    |   movel([0.065962, -1.378345, -2.576120, -0.757924, 1.570796, 1.636759],accel_mss,speed_ms,0,blend_radius_m)
    |   speed_ms = 0.007
    |   movel([0.065737, -1.378110, -2.576285, -0.757994, 1.570796, 1.636533],accel_mss,speed_ms,0,blend_radius_m)
    |   movel([0.065748, -1.377418, -2.576770, -0.758201, 1.570796, 1.636545],accel_mss,speed_ms,0,blend_radius_m)
    |   movel([0.065782, -1.376692, -2.577278, -0.758419, 1.570796, 1.636578],accel_mss,speed_ms,0,blend_radius_m)
    |   movel([0.066186, -1.376388, -2.577490, -0.758511, 1.570796, 1.636982],accel_mss,speed_ms,0,blend_radius_m)
    |   movel([0.067252, -1.376135, -2.577667, -0.758587, 1.570796, 1.638048],accel_mss,speed_ms,0,blend_radius_m)
    |   movel([0.068316, -1.375910, -2.577824, -0.758655, 1.570796, 1.639113],accel_mss,speed_ms,0,blend_radius_m)
    |   movel([0.068585, -1.375943, -2.577801, -0.758645, 1.570796, 1.639381],accel_mss,speed_ms,0,blend_radius_m)
    |   movel([0.068684, -1.376248, -2.577588, -0.758553, 1.570796, 1.639480],accel_mss,speed_ms,0,blend_radius_m)
    |   movel([0.068626, -1.376569, -2.577364, -0.758456, 1.570796, 1.639422],accel_mss,speed_ms,0,blend_radius_m)
    |   movel([0.068470, -1.377126, -2.576974, -0.758289, 1.570796, 1.639267],accel_mss,speed_ms,0,blend_radius_m)
    |   movel([0.068277, -1.377389, -2.576790, -0.758210, 1.570796, 1.639073],accel_mss,speed_ms,0,blend_radius_m)
    |   movel([0.067750, -1.377691, -2.576579, -0.758120, 1.570796, 1.638546],accel_mss,speed_ms,0,blend_radius_m)
    |   movel([0.067148, -1.377954, -2.576394, -0.758041, 1.570796, 1.637944],accel_mss,speed_ms,0,blend_radius_m)
    |   movel([0.066517, -1.378181, -2.576235, -0.757973, 1.570796, 1.637313],accel_mss,speed_ms,0,blend_radius_m)
    |   movel([0.065962, -1.378345, -2.576120, -0.757924, 1.570796, 1.636759],accel_mss,speed_ms,0,blend_radius_m)
    |   speed_ms = 0.003
    |   movel([0.065962, -1.365252, -2.570091, -0.777046, 1.570796, 1.636759],accel_mss,speed_ms,0,blend_radius_m)
    |   speed_ms = 1.000
    |   movel([0.065962, -1.340154, -2.557638, -0.814597, 1.570796, 1.636759],accel_mss,speed_ms,0,blend_radius_m)
    |   movel([0.067314, -1.337303, -2.559523, -0.815563, 1.570796, 1.638110],accel_mss,speed_ms,0,blend_radius_m)
    |   movel([0.067314, -1.362450, -2.572012, -0.777926, 1.570796, 1.638110],accel_mss,speed_ms,0,blend_radius_m)
    |   speed_ms = 0.003
    |   movel([0.067314, -1.372257, -2.576561, -0.763571, 1.570796, 1.638110],accel_mss,speed_ms,0,blend_radius_m)
    |   speed_ms = 0.007
    |   movel([0.067188, -1.372005, -2.576736, -0.763648, 1.570796, 1.637984],accel_mss,speed_ms,0,blend_radius_m)
    |   movel([0.067191, -1.371585, -2.577027, -0.763777, 1.570796, 1.637988],accel_mss,speed_ms,0,blend_radius_m)
    |   movel([0.067248, -1.370744, -2.577609, -0.764035, 1.570796, 1.638044],accel_mss,speed_ms,0,blend_radius_m)
    |   movel([0.067309, -1.370030, -2.578103, -0.764256, 1.570796, 1.638105],accel_mss,speed_ms,0,blend_radius_m)
    |   movel([0.067374, -1.369514, -2.578460, -0.764415, 1.570796, 1.638171],accel_mss,speed_ms,0,blend_radius_m)
    |   movel([0.067446, -1.369137, -2.578720, -0.764532, 1.570796, 1.638242],accel_mss,speed_ms,0,blend_radius_m)
    |   movel([0.067665, -1.368841, -2.578924, -0.764624, 1.570796, 1.638462],accel_mss,speed_ms,0,blend_radius_m)
    |   movel([0.067820, -1.368984, -2.578825, -0.764580, 1.570796, 1.638616],accel_mss,speed_ms,0,blend_radius_m)
    |   movel([0.067982, -1.369133, -2.578722, -0.764534, 1.570796, 1.638778],accel_mss,speed_ms,0,blend_radius_m)
    |   movel([0.067952, -1.369386, -2.578548, -0.764455, 1.570796, 1.638748],accel_mss,speed_ms,0,blend_radius_m)
    |   movel([0.067835, -1.370008, -2.578118, -0.764263, 1.570796, 1.638632],accel_mss,speed_ms,0,blend_radius_m)
    |   movel([0.067755, -1.370486, -2.577788, -0.764115, 1.570796, 1.638552],accel_mss,speed_ms,0,blend_radius_m)
    |   movel([0.067679, -1.370980, -2.577446, -0.763963, 1.570796, 1.638475],accel_mss,speed_ms,0,blend_radius_m)
    |   movel([0.067578, -1.371604, -2.577014, -0.763771, 1.570796, 1.638374],accel_mss,speed_ms,0,blend_radius_m)
    |   movel([0.067495, -1.371960, -2.576767, -0.763662, 1.570796, 1.638292],accel_mss,speed_ms,0,blend_radius_m)
    |   movel([0.067314, -1.372257, -2.576561, -0.763571, 1.570796, 1.638110],accel_mss,speed_ms,0,blend_radius_m)
    |   speed_ms = 0.003
    |   movel([0.067314, -1.375572, -2.578060, -0.758757, 1.570796, 1.638110],accel_mss,speed_ms,0,blend_radius_m)
    |   speed_ms = 0.007
    |   movel([0.067188, -1.375320, -2.578236, -0.758833, 1.570796, 1.637984],accel_mss,speed_ms,0,blend_radius_m)
    |   movel([0.067191, -1.374902, -2.578527, -0.758960, 1.570796, 1.637988],accel_mss,speed_ms,0,blend_radius_m)
    |   movel([0.067248, -1.374063, -2.579111, -0.759215, 1.570796, 1.638044],accel_mss,speed_ms,0,blend_radius_m)
    |   movel([0.067309, -1.373351, -2.579606, -0.759432, 1.570796, 1.638105],accel_mss,speed_ms,0,blend_radius_m)
    |   movel([0.067374, -1.372836, -2.579964, -0.759589, 1.570796, 1.638171],accel_mss,speed_ms,0,blend_radius_m)
    |   movel([0.067446, -1.372460, -2.580224, -0.759705, 1.570796, 1.638242],accel_mss,speed_ms,0,blend_radius_m)
    |   movel([0.067665, -1.372165, -2.580429, -0.759795, 1.570796, 1.638462],accel_mss,speed_ms,0,blend_radius_m)
    |   movel([0.067820, -1.372308, -2.580330, -0.759751, 1.570796, 1.638616],accel_mss,speed_ms,0,blend_radius_m)
    |   movel([0.067982, -1.372456, -2.580227, -0.759706, 1.570796, 1.638778],accel_mss,speed_ms,0,blend_radius_m)
    |   movel([0.067952, -1.372709, -2.580052, -0.759628, 1.570796, 1.638748],accel_mss,speed_ms,0,blend_radius_m)
    |   movel([0.067835, -1.373329, -2.579621, -0.759439, 1.570796, 1.638632],accel_mss,speed_ms,0,blend_radius_m)
    |   movel([0.067755, -1.373806, -2.579290, -0.759293, 1.570796, 1.638552],accel_mss,speed_ms,0,blend_radius_m)
    |   movel([0.067679, -1.374299, -2.578947, -0.759143, 1.570796, 1.638475],accel_mss,speed_ms,0,blend_radius_m)
    |   movel([0.067578, -1.374921, -2.578514, -0.758954, 1.570796, 1.638374],accel_mss,speed_ms,0,blend_radius_m)
    |   movel([0.067495, -1.375275, -2.578267, -0.758847, 1.570796, 1.638292],accel_mss,speed_ms,0,blend_radius_m)
    |   movel([0.067314, -1.375572, -2.578060, -0.758757, 1.570796, 1.638110],accel_mss,speed_ms,0,blend_radius_m)
    |   speed_ms = 0.003
    |   movel([0.067314, -1.362450, -2.572012, -0.777926, 1.570796, 1.638110],accel_mss,speed_ms,0,blend_radius_m)
    |   speed_ms = 1.000
    |   movel([0.067314, -1.337303, -2.559523, -0.815563, 1.570796, 1.638110],accel_mss,speed_ms,0,blend_radius_m)
    |   movel([0.067891, -1.337281, -2.559537, -0.815570, 1.570796, 1.638687],accel_mss,speed_ms,0,blend_radius_m)
    |   movel([0.067891, -1.362429, -2.572027, -0.777933, 1.570796, 1.638687],accel_mss,speed_ms,0,blend_radius_m)
    |   speed_ms = 0.003
    |   movel([0.067891, -1.372236, -2.576575, -0.763578, 1.570796, 1.638687],accel_mss,speed_ms,0,blend_radius_m)
    |   speed_ms = 0.007
    |   movel([0.068086, -1.370934, -2.577478, -0.763977, 1.570796, 1.638882],accel_mss,speed_ms,0,blend_radius_m)
    |   movel([0.068314, -1.369498, -2.578470, -0.764420, 1.570796, 1.639111],accel_mss,speed_ms,0,blend_radius_m)
    |   movel([0.068455, -1.368883, -2.578895, -0.764611, 1.570796, 1.639251],accel_mss,speed_ms,0,blend_radius_m)
    |   movel([0.068616, -1.368544, -2.579128, -0.764716, 1.570796, 1.639412],accel_mss,speed_ms,0,blend_radius_m)
    |   movel([0.068856, -1.368334, -2.579273, -0.764782, 1.570796, 1.639652],accel_mss,speed_ms,0,blend_radius_m)
    |   movel([0.069268, -1.367988, -2.579511, -0.764890, 1.570796, 1.640065],accel_mss,speed_ms,0,blend_radius_m)
    |   movel([0.069506, -1.367501, -2.579846, -0.765042, 1.570796, 1.640303],accel_mss,speed_ms,0,blend_radius_m)
    |   movel([0.069487, -1.367063, -2.580147, -0.765179, 1.570796, 1.640284],accel_mss,speed_ms,0,blend_radius_m)
    |   movel([0.069206, -1.366852, -2.580292, -0.765245, 1.570796, 1.640003],accel_mss,speed_ms,0,blend_radius_m)
    |   movel([0.068881, -1.366852, -2.580292, -0.765245, 1.570796, 1.639677],accel_mss,speed_ms,0,blend_radius_m)
    |   movel([0.068537, -1.367087, -2.580131, -0.765171, 1.570796, 1.639333],accel_mss,speed_ms,0,blend_radius_m)
    |   movel([0.068259, -1.367393, -2.579920, -0.765076, 1.570796, 1.639055],accel_mss,speed_ms,0,blend_radius_m)
    |   movel([0.068159, -1.367743, -2.579680, -0.764966, 1.570796, 1.638956],accel_mss,speed_ms,0,blend_radius_m)
    |   movel([0.068095, -1.368023, -2.579487, -0.764879, 1.570796, 1.638891],accel_mss,speed_ms,0,blend_radius_m)
    |   movel([0.067951, -1.368268, -2.579319, -0.764803, 1.570796, 1.638748],accel_mss,speed_ms,0,blend_radius_m)
    |   movel([0.067551, -1.368495, -2.579162, -0.764732, 1.570796, 1.638348],accel_mss,speed_ms,0,blend_radius_m)
    |   movel([0.067363, -1.368371, -2.579248, -0.764770, 1.570796, 1.638159],accel_mss,speed_ms,0,blend_radius_m)
    |   movel([0.067160, -1.368082, -2.579447, -0.764860, 1.570796, 1.637956],accel_mss,speed_ms,0,blend_radius_m)
    |   movel([0.066968, -1.367808, -2.579635, -0.764946, 1.570796, 1.637764],accel_mss,speed_ms,0,blend_radius_m)
    |   movel([0.066743, -1.367664, -2.579734, -0.764991, 1.570796, 1.637539],accel_mss,speed_ms,0,blend_radius_m)
    |   movel([0.066454, -1.367638, -2.579752, -0.764999, 1.570796, 1.637251],accel_mss,speed_ms,0,blend_radius_m)
    |   movel([0.066073, -1.367717, -2.579698, -0.764974, 1.570796, 1.636869],accel_mss,speed_ms,0,blend_radius_m)
    |   movel([0.065765, -1.367878, -2.579587, -0.764924, 1.570796, 1.636562],accel_mss,speed_ms,0,blend_radius_m)
    |   movel([0.065486, -1.368148, -2.579401, -0.764840, 1.570796, 1.636282],accel_mss,speed_ms,0,blend_radius_m)
    |   movel([0.065298, -1.368462, -2.579185, -0.764742, 1.570796, 1.636095],accel_mss,speed_ms,0,blend_radius_m)
    |   movel([0.065249, -1.368750, -2.578987, -0.764653, 1.570796, 1.636045],accel_mss,speed_ms,0,blend_radius_m)
    |   movel([0.065355, -1.368924, -2.578866, -0.764598, 1.570796, 1.636151],accel_mss,speed_ms,0,blend_radius_m)
    |   movel([0.065666, -1.369073, -2.578764, -0.764552, 1.570796, 1.636462],accel_mss,speed_ms,0,blend_radius_m)
    |   movel([0.066034, -1.369155, -2.578708, -0.764527, 1.570796, 1.636830],accel_mss,speed_ms,0,blend_radius_m)
    |   movel([0.066342, -1.369120, -2.578732, -0.764538, 1.570796, 1.637138],accel_mss,speed_ms,0,blend_radius_m)
    |   movel([0.066688, -1.369137, -2.578720, -0.764532, 1.570796, 1.637484],accel_mss,speed_ms,0,blend_radius_m)
    |   movel([0.066870, -1.369408, -2.578532, -0.764448, 1.570796, 1.637666],accel_mss,speed_ms,0,blend_radius_m)
    |   movel([0.066903, -1.370060, -2.578083, -0.764247, 1.570796, 1.637699],accel_mss,speed_ms,0,blend_radius_m)
    |   movel([0.066779, -1.371453, -2.577118, -0.763817, 1.570796, 1.637575],accel_mss,speed_ms,0,blend_radius_m)
    |   movel([0.066708, -1.372078, -2.576685, -0.763626, 1.570796, 1.637504],accel_mss,speed_ms,0,blend_radius_m)
    |   movel([0.066649, -1.372354, -2.576493, -0.763541, 1.570796, 1.637446],accel_mss,speed_ms,0,blend_radius_m)
    |   movel([0.066450, -1.372560, -2.576351, -0.763479, 1.570796, 1.637247],accel_mss,speed_ms,0,blend_radius_m)
    |   movel([0.066231, -1.372466, -2.576416, -0.763507, 1.570796, 1.637027],accel_mss,speed_ms,0,blend_radius_m)
    |   movel([0.066132, -1.372239, -2.576573, -0.763577, 1.570796, 1.636928],accel_mss,speed_ms,0,blend_radius_m)
    |   movel([0.065933, -1.372130, -2.576649, -0.763610, 1.570796, 1.636729],accel_mss,speed_ms,0,blend_radius_m)
    |   movel([0.065974, -1.371889, -2.576816, -0.763684, 1.570796, 1.636770],accel_mss,speed_ms,0,blend_radius_m)
    |   movel([0.065993, -1.371608, -2.577011, -0.763770, 1.570796, 1.636789],accel_mss,speed_ms,0,blend_radius_m)
    |   movel([0.065755, -1.371549, -2.577052, -0.763788, 1.570796, 1.636552],accel_mss,speed_ms,0,blend_radius_m)
    |   movel([0.065388, -1.371592, -2.577022, -0.763775, 1.570796, 1.636185],accel_mss,speed_ms,0,blend_radius_m)
    |   movel([0.064410, -1.371541, -2.577057, -0.763790, 1.570796, 1.635206],accel_mss,speed_ms,0,blend_radius_m)
    |   movel([0.063662, -1.371220, -2.577280, -0.763889, 1.570796, 1.634458],accel_mss,speed_ms,0,blend_radius_m)
    |   movel([0.063073, -1.370714, -2.577630, -0.764045, 1.570796, 1.633869],accel_mss,speed_ms,0,blend_radius_m)
    |   movel([0.062754, -1.370096, -2.578057, -0.764235, 1.570796, 1.633550],accel_mss,speed_ms,0,blend_radius_m)
    |   movel([0.062718, -1.369302, -2.578606, -0.764481, 1.570796, 1.633515],accel_mss,speed_ms,0,blend_radius_m)
    |   movel([0.062983, -1.368306, -2.579293, -0.764791, 1.570796, 1.633779],accel_mss,speed_ms,0,blend_radius_m)
    |   movel([0.063493, -1.367264, -2.580009, -0.765116, 1.570796, 1.634289],accel_mss,speed_ms,0,blend_radius_m)
    |   movel([0.064187, -1.366327, -2.580653, -0.765410, 1.570796, 1.634984],accel_mss,speed_ms,0,blend_radius_m)
    |   movel([0.064468, -1.366042, -2.580848, -0.765499, 1.570796, 1.635264],accel_mss,speed_ms,0,blend_radius_m)
    |   movel([0.064844, -1.365705, -2.581079, -0.765605, 1.570796, 1.635641],accel_mss,speed_ms,0,blend_radius_m)
    |   movel([0.065259, -1.365367, -2.581310, -0.765712, 1.570796, 1.636055],accel_mss,speed_ms,0,blend_radius_m)
    |   movel([0.065655, -1.365077, -2.581508, -0.765803, 1.570796, 1.636451],accel_mss,speed_ms,0,blend_radius_m)
    |   movel([0.066240, -1.364690, -2.581773, -0.765926, 1.570796, 1.637037],accel_mss,speed_ms,0,blend_radius_m)
    |   movel([0.066630, -1.364481, -2.581916, -0.765992, 1.570796, 1.637427],accel_mss,speed_ms,0,blend_radius_m)
    |   movel([0.067072, -1.364316, -2.582029, -0.766044, 1.570796, 1.637868],accel_mss,speed_ms,0,blend_radius_m)
    |   movel([0.067932, -1.364064, -2.582200, -0.766124, 1.570796, 1.638728],accel_mss,speed_ms,0,blend_radius_m)
    |   movel([0.068629, -1.363881, -2.582325, -0.766182, 1.570796, 1.639426],accel_mss,speed_ms,0,blend_radius_m)
    |   movel([0.069134, -1.363776, -2.582397, -0.766216, 1.570796, 1.639930],accel_mss,speed_ms,0,blend_radius_m)
    |   movel([0.069542, -1.363727, -2.582430, -0.766231, 1.570796, 1.640338],accel_mss,speed_ms,0,blend_radius_m)
    |   movel([0.069913, -1.363729, -2.582429, -0.766231, 1.570796, 1.640709],accel_mss,speed_ms,0,blend_radius_m)
    |   movel([0.070682, -1.363828, -2.582362, -0.766199, 1.570796, 1.641478],accel_mss,speed_ms,0,blend_radius_m)
    |   movel([0.071270, -1.364006, -2.582240, -0.766143, 1.570796, 1.642066],accel_mss,speed_ms,0,blend_radius_m)
    |   movel([0.071742, -1.364286, -2.582049, -0.766054, 1.570796, 1.642538],accel_mss,speed_ms,0,blend_radius_m)
    |   movel([0.072153, -1.364697, -2.581768, -0.765924, 1.570796, 1.642949],accel_mss,speed_ms,0,blend_radius_m)
    |   movel([0.072432, -1.365078, -2.581508, -0.765803, 1.570796, 1.643228],accel_mss,speed_ms,0,blend_radius_m)
    |   movel([0.072562, -1.365356, -2.581318, -0.765716, 1.570796, 1.643358],accel_mss,speed_ms,0,blend_radius_m)
    |   movel([0.072615, -1.365695, -2.581085, -0.765608, 1.570796, 1.643412],accel_mss,speed_ms,0,blend_radius_m)
    |   movel([0.072625, -1.366311, -2.580663, -0.765415, 1.570796, 1.643422],accel_mss,speed_ms,0,blend_radius_m)
    |   movel([0.072624, -1.366703, -2.580394, -0.765292, 1.570796, 1.643421],accel_mss,speed_ms,0,blend_radius_m)
    |   movel([0.072626, -1.367039, -2.580163, -0.765186, 1.570796, 1.643422],accel_mss,speed_ms,0,blend_radius_m)
    |   movel([0.072628, -1.367330, -2.579964, -0.765095, 1.570796, 1.643425],accel_mss,speed_ms,0,blend_radius_m)
    |   movel([0.072329, -1.367646, -2.579746, -0.764996, 1.570796, 1.643125],accel_mss,speed_ms,0,blend_radius_m)
    |   movel([0.072081, -1.368084, -2.579445, -0.764860, 1.570796, 1.642878],accel_mss,speed_ms,0,blend_radius_m)
    |   movel([0.071908, -1.368353, -2.579260, -0.764776, 1.570796, 1.642704],accel_mss,speed_ms,0,blend_radius_m)
    |   movel([0.071728, -1.368608, -2.579084, -0.764697, 1.570796, 1.642524],accel_mss,speed_ms,0,blend_radius_m)
    |   movel([0.071129, -1.369231, -2.578655, -0.764503, 1.570796, 1.641925],accel_mss,speed_ms,0,blend_radius_m)
    |   movel([0.070532, -1.369679, -2.578346, -0.764364, 1.570796, 1.641329],accel_mss,speed_ms,0,blend_radius_m)
    |   movel([0.069917, -1.370062, -2.578081, -0.764246, 1.570796, 1.640713],accel_mss,speed_ms,0,blend_radius_m)
    |   movel([0.069427, -1.370278, -2.577932, -0.764179, 1.570796, 1.640223],accel_mss,speed_ms,0,blend_radius_m)
    |   movel([0.069053, -1.370439, -2.577821, -0.764130, 1.570796, 1.639849],accel_mss,speed_ms,0,blend_radius_m)
    |   movel([0.068800, -1.370627, -2.577690, -0.764071, 1.570796, 1.639597],accel_mss,speed_ms,0,blend_radius_m)
    |   movel([0.068643, -1.370899, -2.577502, -0.763988, 1.570796, 1.639439],accel_mss,speed_ms,0,blend_radius_m)
    |   movel([0.068529, -1.371298, -2.577226, -0.763865, 1.570796, 1.639325],accel_mss,speed_ms,0,blend_radius_m)
    |   movel([0.068476, -1.371655, -2.576978, -0.763755, 1.570796, 1.639272],accel_mss,speed_ms,0,blend_radius_m)
    |   movel([0.068694, -1.371767, -2.576901, -0.763721, 1.570796, 1.639490],accel_mss,speed_ms,0,blend_radius_m)
    |   movel([0.068466, -1.372049, -2.576705, -0.763635, 1.570796, 1.639263],accel_mss,speed_ms,0,blend_radius_m)
    |   movel([0.067891, -1.372236, -2.576575, -0.763578, 1.570796, 1.638687],accel_mss,speed_ms,0,blend_radius_m)
    |   speed_ms = 0.003
    |   movel([0.067891, -1.375551, -2.578075, -0.758763, 1.570796, 1.638687],accel_mss,speed_ms,0,blend_radius_m)
    |   speed_ms = 0.007
    |   movel([0.068086, -1.374253, -2.578979, -0.759157, 1.570796, 1.638882],accel_mss,speed_ms,0,blend_radius_m)
    |   movel([0.068314, -1.372821, -2.579974, -0.759594, 1.570796, 1.639111],accel_mss,speed_ms,0,blend_radius_m)
    |   movel([0.068455, -1.372207, -2.580399, -0.759782, 1.570796, 1.639251],accel_mss,speed_ms,0,blend_radius_m)
    |   movel([0.068616, -1.371869, -2.580634, -0.759886, 1.570796, 1.639412],accel_mss,speed_ms,0,blend_radius_m)
    |   movel([0.068856, -1.371659, -2.580779, -0.759951, 1.570796, 1.639652],accel_mss,speed_ms,0,blend_radius_m)
    |   movel([0.069268, -1.371315, -2.581018, -0.760057, 1.570796, 1.640065],accel_mss,speed_ms,0,blend_radius_m)
    |   movel([0.069506, -1.370829, -2.581353, -0.760207, 1.570796, 1.640303],accel_mss,speed_ms,0,blend_radius_m)
    |   movel([0.069487, -1.370391, -2.581655, -0.760342, 1.570796, 1.640284],accel_mss,speed_ms,0,blend_radius_m)
    |   movel([0.069206, -1.370181, -2.581800, -0.760407, 1.570796, 1.640003],accel_mss,speed_ms,0,blend_radius_m)
    |   movel([0.068881, -1.370181, -2.581801, -0.760407, 1.570796, 1.639677],accel_mss,speed_ms,0,blend_radius_m)
    |   movel([0.068537, -1.370416, -2.581639, -0.760335, 1.570796, 1.639333],accel_mss,speed_ms,0,blend_radius_m)
    |   movel([0.068259, -1.370721, -2.581428, -0.760240, 1.570796, 1.639055],accel_mss,speed_ms,0,blend_radius_m)
    |   movel([0.068159, -1.371070, -2.581186, -0.760132, 1.570796, 1.638956],accel_mss,speed_ms,0,blend_radius_m)
    |   movel([0.068095, -1.371349, -2.580994, -0.760046, 1.570796, 1.638891],accel_mss,speed_ms,0,blend_radius_m)
    |   movel([0.067951, -1.371593, -2.580825, -0.759971, 1.570796, 1.638748],accel_mss,speed_ms,0,blend_radius_m)
    |   movel([0.067551, -1.371820, -2.580668, -0.759901, 1.570796, 1.638348],accel_mss,speed_ms,0,blend_radius_m)
    |   movel([0.067363, -1.371696, -2.580753, -0.759939, 1.570796, 1.638159],accel_mss,speed_ms,0,blend_radius_m)
    |   movel([0.067160, -1.371408, -2.580953, -0.760028, 1.570796, 1.637956],accel_mss,speed_ms,0,blend_radius_m)
    |   movel([0.066968, -1.371135, -2.581142, -0.760112, 1.570796, 1.637764],accel_mss,speed_ms,0,blend_radius_m)
    |   movel([0.066743, -1.370991, -2.581241, -0.760157, 1.570796, 1.637539],accel_mss,speed_ms,0,blend_radius_m)
    |   movel([0.066454, -1.370965, -2.581259, -0.760165, 1.570796, 1.637251],accel_mss,speed_ms,0,blend_radius_m)
    |   movel([0.066073, -1.371044, -2.581205, -0.760140, 1.570796, 1.636869],accel_mss,speed_ms,0,blend_radius_m)
    |   movel([0.065765, -1.371204, -2.581094, -0.760091, 1.570796, 1.636562],accel_mss,speed_ms,0,blend_radius_m)
    |   movel([0.065486, -1.371474, -2.580907, -0.760008, 1.570796, 1.636282],accel_mss,speed_ms,0,blend_radius_m)
    |   movel([0.065298, -1.371787, -2.580690, -0.759911, 1.570796, 1.636095],accel_mss,speed_ms,0,blend_radius_m)
    |   movel([0.065249, -1.372074, -2.580492, -0.759823, 1.570796, 1.636045],accel_mss,speed_ms,0,blend_radius_m)
    |   movel([0.065355, -1.372248, -2.580371, -0.759770, 1.570796, 1.636151],accel_mss,speed_ms,0,blend_radius_m)
    |   movel([0.065666, -1.372396, -2.580268, -0.759724, 1.570796, 1.636462],accel_mss,speed_ms,0,blend_radius_m)
    |   movel([0.066034, -1.372478, -2.580212, -0.759699, 1.570796, 1.636830],accel_mss,speed_ms,0,blend_radius_m)
    |   movel([0.066342, -1.372443, -2.580236, -0.759710, 1.570796, 1.637138],accel_mss,speed_ms,0,blend_radius_m)
    |   movel([0.066688, -1.372460, -2.580224, -0.759705, 1.570796, 1.637484],accel_mss,speed_ms,0,blend_radius_m)
    |   movel([0.066870, -1.372731, -2.580036, -0.759622, 1.570796, 1.637666],accel_mss,speed_ms,0,blend_radius_m)
    |   movel([0.066903, -1.373380, -2.579586, -0.759423, 1.570796, 1.637699],accel_mss,speed_ms,0,blend_radius_m)
    |   movel([0.066779, -1.374771, -2.578619, -0.759000, 1.570796, 1.637575],accel_mss,speed_ms,0,blend_radius_m)
    |   movel([0.066708, -1.375394, -2.578185, -0.758811, 1.570796, 1.637504],accel_mss,speed_ms,0,blend_radius_m)
    |   movel([0.066649, -1.375669, -2.577992, -0.758728, 1.570796, 1.637446],accel_mss,speed_ms,0,blend_radius_m)
    |   movel([0.066450, -1.375874, -2.577849, -0.758666, 1.570796, 1.637247],accel_mss,speed_ms,0,blend_radius_m)
    |   movel([0.066231, -1.375780, -2.577915, -0.758694, 1.570796, 1.637027],accel_mss,speed_ms,0,blend_radius_m)
    |   movel([0.066132, -1.375554, -2.578073, -0.758762, 1.570796, 1.636928],accel_mss,speed_ms,0,blend_radius_m)
    |   movel([0.065933, -1.375445, -2.578149, -0.758795, 1.570796, 1.636729],accel_mss,speed_ms,0,blend_radius_m)
    |   movel([0.065974, -1.375205, -2.578316, -0.758868, 1.570796, 1.636770],accel_mss,speed_ms,0,blend_radius_m)
    |   movel([0.065993, -1.374925, -2.578511, -0.758953, 1.570796, 1.636789],accel_mss,speed_ms,0,blend_radius_m)
    |   movel([0.065755, -1.374866, -2.578552, -0.758971, 1.570796, 1.636552],accel_mss,speed_ms,0,blend_radius_m)
    |   movel([0.065388, -1.374909, -2.578523, -0.758958, 1.570796, 1.636185],accel_mss,speed_ms,0,blend_radius_m)
    |   movel([0.064410, -1.374858, -2.578558, -0.758973, 1.570796, 1.635206],accel_mss,speed_ms,0,blend_radius_m)
    |   movel([0.063662, -1.374538, -2.578781, -0.759070, 1.570796, 1.634458],accel_mss,speed_ms,0,blend_radius_m)
    |   movel([0.063073, -1.374033, -2.579132, -0.759224, 1.570796, 1.633869],accel_mss,speed_ms,0,blend_radius_m)
    |   movel([0.062754, -1.373417, -2.579560, -0.759412, 1.570796, 1.633550],accel_mss,speed_ms,0,blend_radius_m)
    |   movel([0.062718, -1.372625, -2.580110, -0.759654, 1.570796, 1.633515],accel_mss,speed_ms,0,blend_radius_m)
    |   movel([0.062983, -1.371631, -2.580799, -0.759959, 1.570796, 1.633779],accel_mss,speed_ms,0,blend_radius_m)
    |   movel([0.063493, -1.370592, -2.581517, -0.760280, 1.570796, 1.634289],accel_mss,speed_ms,0,blend_radius_m)
    |   movel([0.064187, -1.369657, -2.582162, -0.760570, 1.570796, 1.634984],accel_mss,speed_ms,0,blend_radius_m)
    |   movel([0.064468, -1.369373, -2.582357, -0.760658, 1.570796, 1.635264],accel_mss,speed_ms,0,blend_radius_m)
    |   movel([0.064844, -1.369037, -2.582589, -0.760763, 1.570796, 1.635641],accel_mss,speed_ms,0,blend_radius_m)
    |   movel([0.065259, -1.368700, -2.582821, -0.760868, 1.570796, 1.636055],accel_mss,speed_ms,0,blend_radius_m)
    |   movel([0.065655, -1.368412, -2.583019, -0.760958, 1.570796, 1.636451],accel_mss,speed_ms,0,blend_radius_m)
    |   movel([0.066240, -1.368025, -2.583285, -0.761079, 1.570796, 1.637037],accel_mss,speed_ms,0,blend_radius_m)
    |   movel([0.066630, -1.367817, -2.583428, -0.761144, 1.570796, 1.637427],accel_mss,speed_ms,0,blend_radius_m)
    |   movel([0.067072, -1.367652, -2.583541, -0.761196, 1.570796, 1.637868],accel_mss,speed_ms,0,blend_radius_m)
    |   movel([0.067932, -1.367401, -2.583713, -0.761275, 1.570796, 1.638728],accel_mss,speed_ms,0,blend_radius_m)
    |   movel([0.068629, -1.367218, -2.583839, -0.761332, 1.570796, 1.639426],accel_mss,speed_ms,0,blend_radius_m)
    |   movel([0.069134, -1.367114, -2.583910, -0.761365, 1.570796, 1.639930],accel_mss,speed_ms,0,blend_radius_m)
    |   movel([0.069542, -1.367065, -2.583944, -0.761380, 1.570796, 1.640338],accel_mss,speed_ms,0,blend_radius_m)
    |   movel([0.069913, -1.367066, -2.583943, -0.761380, 1.570796, 1.640709],accel_mss,speed_ms,0,blend_radius_m)
    |   movel([0.070682, -1.367165, -2.583875, -0.761349, 1.570796, 1.641478],accel_mss,speed_ms,0,blend_radius_m)
    |   movel([0.071270, -1.367343, -2.583753, -0.761293, 1.570796, 1.642066],accel_mss,speed_ms,0,blend_radius_m)
    |   movel([0.071742, -1.367622, -2.583561, -0.761205, 1.570796, 1.642538],accel_mss,speed_ms,0,blend_radius_m)
    |   movel([0.072153, -1.368032, -2.583280, -0.761077, 1.570796, 1.642949],accel_mss,speed_ms,0,blend_radius_m)
    |   movel([0.072432, -1.368412, -2.583019, -0.760958, 1.570796, 1.643228],accel_mss,speed_ms,0,blend_radius_m)
    |   movel([0.072562, -1.368689, -2.582828, -0.760872, 1.570796, 1.643358],accel_mss,speed_ms,0,blend_radius_m)
    |   movel([0.072615, -1.369028, -2.582595, -0.760766, 1.570796, 1.643412],accel_mss,speed_ms,0,blend_radius_m)
    |   movel([0.072625, -1.369642, -2.582173, -0.760575, 1.570796, 1.643422],accel_mss,speed_ms,0,blend_radius_m)
    |   movel([0.072624, -1.370033, -2.581903, -0.760453, 1.570796, 1.643421],accel_mss,speed_ms,0,blend_radius_m)
    |   movel([0.072626, -1.370368, -2.581671, -0.760349, 1.570796, 1.643422],accel_mss,speed_ms,0,blend_radius_m)
    |   movel([0.072628, -1.370658, -2.581471, -0.760260, 1.570796, 1.643425],accel_mss,speed_ms,0,blend_radius_m)
    |   movel([0.072329, -1.370973, -2.581253, -0.760162, 1.570796, 1.643125],accel_mss,speed_ms,0,blend_radius_m)
    |   movel([0.072081, -1.371410, -2.580951, -0.760027, 1.570796, 1.642878],accel_mss,speed_ms,0,blend_radius_m)
    |   movel([0.071908, -1.371678, -2.580766, -0.759945, 1.570796, 1.642704],accel_mss,speed_ms,0,blend_radius_m)
    |   movel([0.071728, -1.371933, -2.580590, -0.759867, 1.570796, 1.642524],accel_mss,speed_ms,0,blend_radius_m)
    |   movel([0.071129, -1.372554, -2.580159, -0.759676, 1.570796, 1.641925],accel_mss,speed_ms,0,blend_radius_m)
    |   movel([0.070532, -1.373001, -2.579849, -0.759539, 1.570796, 1.641329],accel_mss,speed_ms,0,blend_radius_m)
    |   movel([0.069917, -1.373383, -2.579584, -0.759422, 1.570796, 1.640713],accel_mss,speed_ms,0,blend_radius_m)
    |   movel([0.069427, -1.373598, -2.579434, -0.759356, 1.570796, 1.640223],accel_mss,speed_ms,0,blend_radius_m)
    |   movel([0.069053, -1.373758, -2.579323, -0.759308, 1.570796, 1.639849],accel_mss,speed_ms,0,blend_radius_m)
    |   movel([0.068800, -1.373947, -2.579192, -0.759250, 1.570796, 1.639597],accel_mss,speed_ms,0,blend_radius_m)
    |   movel([0.068643, -1.374217, -2.579004, -0.759168, 1.570796, 1.639439],accel_mss,speed_ms,0,blend_radius_m)
    |   movel([0.068529, -1.374615, -2.578727, -0.759047, 1.570796, 1.639325],accel_mss,speed_ms,0,blend_radius_m)
    |   movel([0.068476, -1.374972, -2.578479, -0.758939, 1.570796, 1.639272],accel_mss,speed_ms,0,blend_radius_m)
    |   movel([0.068694, -1.375083, -2.578401, -0.758905, 1.570796, 1.639490],accel_mss,speed_ms,0,blend_radius_m)
    |   movel([0.068466, -1.375365, -2.578205, -0.758820, 1.570796, 1.639263],accel_mss,speed_ms,0,blend_radius_m)
    |   movel([0.067891, -1.375551, -2.578075, -0.758763, 1.570796, 1.638687],accel_mss,speed_ms,0,blend_radius_m)
    |   speed_ms = 0.003
    |   movel([0.067891, -1.362429, -2.572027, -0.777933, 1.570796, 1.638687],accel_mss,speed_ms,0,blend_radius_m)
    |   speed_ms = 1.000
    |   movel([0.067891, -1.337281, -2.559537, -0.815570, 1.570796, 1.638687],accel_mss,speed_ms,0,blend_radius_m)
    |   movel([0.068557, -1.332885, -2.562423, -0.817081, 1.570796, 1.639354],accel_mss,speed_ms,0,blend_radius_m)
    |   movel([0.068557, -1.358109, -2.574969, -0.779311, 1.570796, 1.639354],accel_mss,speed_ms,0,blend_radius_m)
    |   speed_ms = 0.003
    |   movel([0.068557, -1.367949, -2.579538, -0.764902, 1.570796, 1.639354],accel_mss,speed_ms,0,blend_radius_m)
    |   speed_ms = 0.007
    |   movel([0.068577, -1.367549, -2.579813, -0.765027, 1.570796, 1.639373],accel_mss,speed_ms,0,blend_radius_m)
    |   movel([0.068828, -1.367296, -2.579987, -0.765106, 1.570796, 1.639624],accel_mss,speed_ms,0,blend_radius_m)
    |   movel([0.069143, -1.367298, -2.579986, -0.765105, 1.570796, 1.639939],accel_mss,speed_ms,0,blend_radius_m)
    |   movel([0.069072, -1.367533, -2.579824, -0.765032, 1.570796, 1.639868],accel_mss,speed_ms,0,blend_radius_m)
    |   movel([0.068842, -1.367743, -2.579680, -0.764966, 1.570796, 1.639638],accel_mss,speed_ms,0,blend_radius_m)
    |   movel([0.068557, -1.367949, -2.579538, -0.764902, 1.570796, 1.639354],accel_mss,speed_ms,0,blend_radius_m)
    |   speed_ms = 0.003
    |   movel([0.068557, -1.371275, -2.581045, -0.760069, 1.570796, 1.639354],accel_mss,speed_ms,0,blend_radius_m)
    |   speed_ms = 0.007
    |   movel([0.068577, -1.370876, -2.581320, -0.760192, 1.570796, 1.639373],accel_mss,speed_ms,0,blend_radius_m)
    |   movel([0.068828, -1.370624, -2.581495, -0.760270, 1.570796, 1.639624],accel_mss,speed_ms,0,blend_radius_m)
    |   movel([0.069143, -1.370626, -2.581493, -0.760270, 1.570796, 1.639939],accel_mss,speed_ms,0,blend_radius_m)
    |   movel([0.069072, -1.370860, -2.581332, -0.760197, 1.570796, 1.639868],accel_mss,speed_ms,0,blend_radius_m)
    |   movel([0.068842, -1.371070, -2.581187, -0.760132, 1.570796, 1.639638],accel_mss,speed_ms,0,blend_radius_m)
    |   movel([0.068557, -1.371275, -2.581045, -0.760069, 1.570796, 1.639354],accel_mss,speed_ms,0,blend_radius_m)
    |   speed_ms = 0.003
    |   movel([0.068557, -1.358109, -2.574969, -0.779311, 1.570796, 1.639354],accel_mss,speed_ms,0,blend_radius_m)
    |   speed_ms = 1.000
    |   movel([0.068557, -1.332885, -2.562423, -0.817081, 1.570796, 1.639354],accel_mss,speed_ms,0,blend_radius_m)
    |   movel([0.066722, -1.333449, -2.562054, -0.816886, 1.570796, 1.637519],accel_mss,speed_ms,0,blend_radius_m)
    |   movel([0.066722, -1.358664, -2.574592, -0.779133, 1.570796, 1.637519],accel_mss,speed_ms,0,blend_radius_m)
    |   speed_ms = 0.003
    |   movel([0.066722, -1.368499, -2.579159, -0.764730, 1.570796, 1.637519],accel_mss,speed_ms,0,blend_radius_m)
    |   speed_ms = 0.007
    |   movel([0.066563, -1.368732, -2.578999, -0.764658, 1.570796, 1.637359],accel_mss,speed_ms,0,blend_radius_m)
    |   movel([0.066206, -1.368695, -2.579024, -0.764669, 1.570796, 1.637002],accel_mss,speed_ms,0,blend_radius_m)
    |   movel([0.065869, -1.368561, -2.579117, -0.764711, 1.570796, 1.636665],accel_mss,speed_ms,0,blend_radius_m)
    |   movel([0.065944, -1.368236, -2.579341, -0.764812, 1.570796, 1.636740],accel_mss,speed_ms,0,blend_radius_m)
    |   movel([0.066166, -1.368019, -2.579490, -0.764880, 1.570796, 1.636963],accel_mss,speed_ms,0,blend_radius_m)
    |   movel([0.066451, -1.368162, -2.579392, -0.764836, 1.570796, 1.637247],accel_mss,speed_ms,0,blend_radius_m)
    |   movel([0.066639, -1.368330, -2.579276, -0.764783, 1.570796, 1.637435],accel_mss,speed_ms,0,blend_radius_m)
    |   speed_ms = 0.003
    |   movel([0.066722, -1.371824, -2.580665, -0.759900, 1.570796, 1.637519],accel_mss,speed_ms,0,blend_radius_m)
    |   speed_ms = 0.007
    |   movel([0.066563, -1.372056, -2.580504, -0.759829, 1.570796, 1.637359],accel_mss,speed_ms,0,blend_radius_m)
    |   movel([0.066206, -1.372020, -2.580529, -0.759840, 1.570796, 1.637002],accel_mss,speed_ms,0,blend_radius_m)
    |   movel([0.065869, -1.371886, -2.580622, -0.759881, 1.570796, 1.636665],accel_mss,speed_ms,0,blend_radius_m)
    |   movel([0.065944, -1.371562, -2.580847, -0.759981, 1.570796, 1.636740],accel_mss,speed_ms,0,blend_radius_m)
    |   movel([0.066166, -1.371346, -2.580996, -0.760047, 1.570796, 1.636963],accel_mss,speed_ms,0,blend_radius_m)
    |   movel([0.066451, -1.371488, -2.580898, -0.760004, 1.570796, 1.637247],accel_mss,speed_ms,0,blend_radius_m)
    |   movel([0.066639, -1.371655, -2.580782, -0.759952, 1.570796, 1.637435],accel_mss,speed_ms,0,blend_radius_m)
    |   speed_ms = 0.003
    |   movel([0.066722, -1.358664, -2.574592, -0.779133, 1.570796, 1.637519],accel_mss,speed_ms,0,blend_radius_m)
    |   speed_ms = 1.000
    |   movel([0.066722, -1.333449, -2.562054, -0.816886, 1.570796, 1.637519],accel_mss,speed_ms,0,blend_radius_m)
    |   movel([0.065746, -1.318776, -2.571512, -0.822101, 1.570796, 1.636542],accel_mss,speed_ms,0,blend_radius_m)
    |   movel([0.065746, -1.344239, -2.584239, -0.783911, 1.570796, 1.636542],accel_mss,speed_ms,0,blend_radius_m)
    |   speed_ms = 0.003
    |   movel([0.065746, -1.354182, -2.588877, -0.769330, 1.570796, 1.636542],accel_mss,speed_ms,0,blend_radius_m)
    |   speed_ms = 0.007
    |   movel([0.065772, -1.353710, -2.589193, -0.769486, 1.570796, 1.636568],accel_mss,speed_ms,0,blend_radius_m)
    |   movel([0.066112, -1.352862, -2.589759, -0.769768, 1.570796, 1.636908],accel_mss,speed_ms,0,blend_radius_m)
    |   movel([0.067083, -1.350617, -2.591252, -0.770519, 1.570796, 1.637880],accel_mss,speed_ms,0,blend_radius_m)
    |   movel([0.067719, -1.349136, -2.592234, -0.771019, 1.570796, 1.638515],accel_mss,speed_ms,0,blend_radius_m)
    |   movel([0.068073, -1.348257, -2.592815, -0.771317, 1.570796, 1.638869],accel_mss,speed_ms,0,blend_radius_m)
    |   movel([0.068273, -1.347685, -2.593193, -0.771511, 1.570796, 1.639069],accel_mss,speed_ms,0,blend_radius_m)
    |   movel([0.068106, -1.347511, -2.593307, -0.771570, 1.570796, 1.638903],accel_mss,speed_ms,0,blend_radius_m)
    |   movel([0.067773, -1.347577, -2.593264, -0.771548, 1.570796, 1.638570],accel_mss,speed_ms,0,blend_radius_m)
    |   movel([0.067262, -1.347717, -2.593172, -0.771501, 1.570796, 1.638058],accel_mss,speed_ms,0,blend_radius_m)
    |   movel([0.066457, -1.347971, -2.593004, -0.771414, 1.570796, 1.637253],accel_mss,speed_ms,0,blend_radius_m)
    |   movel([0.065785, -1.348180, -2.592866, -0.771343, 1.570796, 1.636581],accel_mss,speed_ms,0,blend_radius_m)
    |   movel([0.065232, -1.348336, -2.592763, -0.771290, 1.570796, 1.636028],accel_mss,speed_ms,0,blend_radius_m)
    |   movel([0.064791, -1.348447, -2.592690, -0.771252, 1.570796, 1.635588],accel_mss,speed_ms,0,blend_radius_m)
    |   movel([0.064973, -1.347487, -2.593324, -0.771579, 1.570796, 1.635770],accel_mss,speed_ms,0,blend_radius_m)
    |   movel([0.065442, -1.346342, -2.594078, -0.771970, 1.570796, 1.636238],accel_mss,speed_ms,0,blend_radius_m)
    |   movel([0.066182, -1.344629, -2.595202, -0.772557, 1.570796, 1.636979],accel_mss,speed_ms,0,blend_radius_m)
    |   movel([0.066820, -1.343178, -2.596152, -0.773059, 1.570796, 1.637617],accel_mss,speed_ms,0,blend_radius_m)
    |   movel([0.067378, -1.341927, -2.596969, -0.773494, 1.570796, 1.638175],accel_mss,speed_ms,0,blend_radius_m)
    |   movel([0.067871, -1.340832, -2.597682, -0.773876, 1.570796, 1.638668],accel_mss,speed_ms,0,blend_radius_m)
    |   movel([0.068273, -1.340444, -2.597934, -0.774011, 1.570796, 1.639070],accel_mss,speed_ms,0,blend_radius_m)
    |   movel([0.070568, -1.339691, -2.598423, -0.774275, 1.570796, 1.641364],accel_mss,speed_ms,0,blend_radius_m)
    |   movel([0.072875, -1.338962, -2.598895, -0.774532, 1.570796, 1.643671],accel_mss,speed_ms,0,blend_radius_m)
    |   movel([0.073115, -1.339033, -2.598849, -0.774507, 1.570796, 1.643911],accel_mss,speed_ms,0,blend_radius_m)
    |   movel([0.072689, -1.339919, -2.598275, -0.774195, 1.570796, 1.643486],accel_mss,speed_ms,0,blend_radius_m)
    |   movel([0.072189, -1.340820, -2.597690, -0.773880, 1.570796, 1.642986],accel_mss,speed_ms,0,blend_radius_m)
    |   movel([0.071589, -1.341857, -2.597014, -0.773518, 1.570796, 1.642385],accel_mss,speed_ms,0,blend_radius_m)
    |   movel([0.070780, -1.343250, -2.596105, -0.773034, 1.570796, 1.641576],accel_mss,speed_ms,0,blend_radius_m)
    |   movel([0.070360, -1.344020, -2.595601, -0.772768, 1.570796, 1.641156],accel_mss,speed_ms,0,blend_radius_m)
    |   movel([0.070135, -1.344497, -2.595289, -0.772603, 1.570796, 1.640931],accel_mss,speed_ms,0,blend_radius_m)
    |   movel([0.070293, -1.344677, -2.595171, -0.772541, 1.570796, 1.641090],accel_mss,speed_ms,0,blend_radius_m)
    |   movel([0.070585, -1.344629, -2.595202, -0.772558, 1.570796, 1.641381],accel_mss,speed_ms,0,blend_radius_m)
    |   movel([0.071041, -1.344508, -2.595281, -0.772599, 1.570796, 1.641837],accel_mss,speed_ms,0,blend_radius_m)
    |   movel([0.071762, -1.344282, -2.595430, -0.772677, 1.570796, 1.642559],accel_mss,speed_ms,0,blend_radius_m)
    |   movel([0.072728, -1.343981, -2.595627, -0.772781, 1.570796, 1.643524],accel_mss,speed_ms,0,blend_radius_m)
    |   movel([0.073151, -1.343887, -2.595689, -0.772814, 1.570796, 1.643947],accel_mss,speed_ms,0,blend_radius_m)
    |   movel([0.073323, -1.344073, -2.595566, -0.772749, 1.570796, 1.644120],accel_mss,speed_ms,0,blend_radius_m)
    |   movel([0.072183, -1.345650, -2.594532, -0.772207, 1.570796, 1.642979],accel_mss,speed_ms,0,blend_radius_m)
    |   movel([0.070974, -1.347290, -2.593453, -0.771646, 1.570796, 1.641770],accel_mss,speed_ms,0,blend_radius_m)
    |   movel([0.069560, -1.349198, -2.592193, -0.770998, 1.570796, 1.640356],accel_mss,speed_ms,0,blend_radius_m)
    |   movel([0.068144, -1.351097, -2.590934, -0.770358, 1.570796, 1.638941],accel_mss,speed_ms,0,blend_radius_m)
    |   movel([0.066928, -1.352699, -2.589867, -0.769822, 1.570796, 1.637725],accel_mss,speed_ms,0,blend_radius_m)
    |   movel([0.065852, -1.354104, -2.588929, -0.769356, 1.570796, 1.636649],accel_mss,speed_ms,0,blend_radius_m)
    |   speed_ms = 0.003
    |   movel([0.065746, -1.357545, -2.590406, -0.764438, 1.570796, 1.636542],accel_mss,speed_ms,0,blend_radius_m)
    |   speed_ms = 0.007
    |   movel([0.065772, -1.357073, -2.590723, -0.764593, 1.570796, 1.636568],accel_mss,speed_ms,0,blend_radius_m)
    |   movel([0.066112, -1.356228, -2.591290, -0.764871, 1.570796, 1.636908],accel_mss,speed_ms,0,blend_radius_m)
    |   movel([0.067083, -1.353989, -2.592787, -0.765613, 1.570796, 1.637880],accel_mss,speed_ms,0,blend_radius_m)
    |   movel([0.067719, -1.352512, -2.593772, -0.766106, 1.570796, 1.638515],accel_mss,speed_ms,0,blend_radius_m)
    |   movel([0.068073, -1.351635, -2.594354, -0.766400, 1.570796, 1.638869],accel_mss,speed_ms,0,blend_radius_m)
    |   movel([0.068273, -1.351064, -2.594733, -0.766592, 1.570796, 1.639069],accel_mss,speed_ms,0,blend_radius_m)
    |   movel([0.068106, -1.350891, -2.594848, -0.766650, 1.570796, 1.638903],accel_mss,speed_ms,0,blend_radius_m)
    |   movel([0.067773, -1.350957, -2.594804, -0.766628, 1.570796, 1.638570],accel_mss,speed_ms,0,blend_radius_m)
    |   movel([0.067262, -1.351096, -2.594712, -0.766581, 1.570796, 1.638058],accel_mss,speed_ms,0,blend_radius_m)
    |   movel([0.066457, -1.351350, -2.594543, -0.766496, 1.570796, 1.637253],accel_mss,speed_ms,0,blend_radius_m)
    |   movel([0.065785, -1.351558, -2.594405, -0.766426, 1.570796, 1.636581],accel_mss,speed_ms,0,blend_radius_m)
    |   movel([0.065232, -1.351714, -2.594302, -0.766373, 1.570796, 1.636028],accel_mss,speed_ms,0,blend_radius_m)
    |   movel([0.064791, -1.351824, -2.594229, -0.766336, 1.570796, 1.635588],accel_mss,speed_ms,0,blend_radius_m)
    |   movel([0.064973, -1.350866, -2.594864, -0.766659, 1.570796, 1.635770],accel_mss,speed_ms,0,blend_radius_m)
    |   movel([0.065442, -1.349724, -2.595620, -0.767045, 1.570796, 1.636238],accel_mss,speed_ms,0,blend_radius_m)
    |   movel([0.066182, -1.348016, -2.596747, -0.767625, 1.570796, 1.636979],accel_mss,speed_ms,0,blend_radius_m)
    |   movel([0.066820, -1.346569, -2.597700, -0.768121, 1.570796, 1.637617],accel_mss,speed_ms,0,blend_radius_m)
    |   movel([0.067378, -1.345321, -2.598518, -0.768550, 1.570796, 1.638175],accel_mss,speed_ms,0,blend_radius_m)
    |   movel([0.067871, -1.344228, -2.599233, -0.768927, 1.570796, 1.638668],accel_mss,speed_ms,0,blend_radius_m)
    |   movel([0.068273, -1.343841, -2.599486, -0.769062, 1.570796, 1.639070],accel_mss,speed_ms,0,blend_radius_m)
    |   movel([0.070568, -1.343090, -2.599976, -0.769323, 1.570796, 1.641364],accel_mss,speed_ms,0,blend_radius_m)
    |   movel([0.072875, -1.342363, -2.600450, -0.769576, 1.570796, 1.643671],accel_mss,speed_ms,0,blend_radius_m)
    |   movel([0.073115, -1.342434, -2.600404, -0.769551, 1.570796, 1.643911],accel_mss,speed_ms,0,blend_radius_m)
    |   movel([0.072689, -1.343318, -2.599828, -0.769243, 1.570796, 1.643486],accel_mss,speed_ms,0,blend_radius_m)
    |   movel([0.072189, -1.344216, -2.599241, -0.768932, 1.570796, 1.642986],accel_mss,speed_ms,0,blend_radius_m)
    |   movel([0.071589, -1.345251, -2.598564, -0.768574, 1.570796, 1.642385],accel_mss,speed_ms,0,blend_radius_m)
    |   movel([0.070780, -1.346641, -2.597652, -0.768096, 1.570796, 1.641576],accel_mss,speed_ms,0,blend_radius_m)
    |   movel([0.070360, -1.347409, -2.597148, -0.767833, 1.570796, 1.641156],accel_mss,speed_ms,0,blend_radius_m)
    |   movel([0.070135, -1.347885, -2.596834, -0.767670, 1.570796, 1.640931],accel_mss,speed_ms,0,blend_radius_m)
    |   movel([0.070293, -1.348064, -2.596716, -0.767609, 1.570796, 1.641090],accel_mss,speed_ms,0,blend_radius_m)
    |   movel([0.070585, -1.348016, -2.596748, -0.767625, 1.570796, 1.641381],accel_mss,speed_ms,0,blend_radius_m)
    |   movel([0.071041, -1.347896, -2.596827, -0.767666, 1.570796, 1.641837],accel_mss,speed_ms,0,blend_radius_m)
    |   movel([0.071762, -1.347670, -2.596975, -0.767743, 1.570796, 1.642559],accel_mss,speed_ms,0,blend_radius_m)
    |   movel([0.072728, -1.347369, -2.597173, -0.767846, 1.570796, 1.643524],accel_mss,speed_ms,0,blend_radius_m)
    |   movel([0.073151, -1.347276, -2.597235, -0.767878, 1.570796, 1.643947],accel_mss,speed_ms,0,blend_radius_m)
    |   movel([0.073323, -1.347462, -2.597113, -0.767815, 1.570796, 1.644120],accel_mss,speed_ms,0,blend_radius_m)
    |   movel([0.072183, -1.349035, -2.596076, -0.767279, 1.570796, 1.642979],accel_mss,speed_ms,0,blend_radius_m)
    |   movel([0.070974, -1.350670, -2.594994, -0.766725, 1.570796, 1.641770],accel_mss,speed_ms,0,blend_radius_m)
    |   movel([0.069560, -1.352574, -2.593730, -0.766085, 1.570796, 1.640356],accel_mss,speed_ms,0,blend_radius_m)
    |   movel([0.068144, -1.354467, -2.592468, -0.765453, 1.570796, 1.638941],accel_mss,speed_ms,0,blend_radius_m)
    |   movel([0.066928, -1.356066, -2.591399, -0.764924, 1.570796, 1.637725],accel_mss,speed_ms,0,blend_radius_m)
    |   movel([0.065852, -1.357467, -2.590459, -0.764463, 1.570796, 1.636649],accel_mss,speed_ms,0,blend_radius_m)
    |   speed_ms = 0.003
    |   movel([0.065746, -1.344239, -2.584239, -0.783911, 1.570796, 1.636542],accel_mss,speed_ms,0,blend_radius_m)
    |   speed_ms = 1.000
    |   movel([0.065746, -1.318776, -2.571512, -0.822101, 1.570796, 1.636542],accel_mss,speed_ms,0,blend_radius_m)
    |   movel([0.081492, -1.289170, -2.589753, -0.833466, 1.570796, 1.652288],accel_mss,speed_ms,0,blend_radius_m)
    |   movel([0.081492, -1.315103, -2.602865, -0.794421, 1.570796, 1.652288],accel_mss,speed_ms,0,blend_radius_m)
    |   speed_ms = 0.003
    |   movel([0.081492, -1.325253, -2.607648, -0.779489, 1.570796, 1.652288],accel_mss,speed_ms,0,blend_radius_m)
    |   speed_ms = 0.007
    |   movel([0.081341, -1.325030, -2.607788, -0.779571, 1.570796, 1.652138],accel_mss,speed_ms,0,blend_radius_m)
    |   movel([0.081467, -1.324183, -2.608320, -0.779886, 1.570796, 1.652263],accel_mss,speed_ms,0,blend_radius_m)
    |   movel([0.081769, -1.322931, -2.609105, -0.780353, 1.570796, 1.652565],accel_mss,speed_ms,0,blend_radius_m)
    |   movel([0.082314, -1.321124, -2.610234, -0.781031, 1.570796, 1.653110],accel_mss,speed_ms,0,blend_radius_m)
    |   movel([0.082603, -1.320135, -2.610851, -0.781404, 1.570796, 1.653400],accel_mss,speed_ms,0,blend_radius_m)
    |   movel([0.082660, -1.319646, -2.611154, -0.781588, 1.570796, 1.653456],accel_mss,speed_ms,0,blend_radius_m)
    |   movel([0.082527, -1.319485, -2.611255, -0.781649, 1.570796, 1.653323],accel_mss,speed_ms,0,blend_radius_m)
    |   movel([0.082236, -1.319545, -2.611217, -0.781627, 1.570796, 1.653033],accel_mss,speed_ms,0,blend_radius_m)
    |   movel([0.081751, -1.319793, -2.611063, -0.781533, 1.570796, 1.652547],accel_mss,speed_ms,0,blend_radius_m)
    |   movel([0.081384, -1.319972, -2.610952, -0.781465, 1.570796, 1.652181],accel_mss,speed_ms,0,blend_radius_m)
    |   movel([0.081002, -1.320156, -2.610837, -0.781396, 1.570796, 1.651798],accel_mss,speed_ms,0,blend_radius_m)
    |   movel([0.080195, -1.320466, -2.610644, -0.781279, 1.570796, 1.650992],accel_mss,speed_ms,0,blend_radius_m)
    |   movel([0.079870, -1.320370, -2.610704, -0.781315, 1.570796, 1.650667],accel_mss,speed_ms,0,blend_radius_m)
    |   movel([0.079791, -1.319865, -2.611018, -0.781506, 1.570796, 1.650588],accel_mss,speed_ms,0,blend_radius_m)
    |   movel([0.079966, -1.317934, -2.612217, -0.782238, 1.570796, 1.650762],accel_mss,speed_ms,0,blend_radius_m)
    |   movel([0.080077, -1.316920, -2.612844, -0.782625, 1.570796, 1.650873],accel_mss,speed_ms,0,blend_radius_m)
    |   movel([0.080182, -1.316146, -2.613323, -0.782921, 1.570796, 1.650979],accel_mss,speed_ms,0,blend_radius_m)
    |   movel([0.080285, -1.315545, -2.613693, -0.783151, 1.570796, 1.651081],accel_mss,speed_ms,0,blend_radius_m)
    |   movel([0.080559, -1.315193, -2.613910, -0.783286, 1.570796, 1.651355],accel_mss,speed_ms,0,blend_radius_m)
    |   movel([0.080916, -1.314988, -2.614036, -0.783365, 1.570796, 1.651713],accel_mss,speed_ms,0,blend_radius_m)
    |   movel([0.081474, -1.314721, -2.614200, -0.783468, 1.570796, 1.652271],accel_mss,speed_ms,0,blend_radius_m)
    |   movel([0.082380, -1.314335, -2.614437, -0.783616, 1.570796, 1.653176],accel_mss,speed_ms,0,blend_radius_m)
    |   movel([0.083212, -1.314002, -2.614642, -0.783745, 1.570796, 1.654008],accel_mss,speed_ms,0,blend_radius_m)
    |   movel([0.083713, -1.313842, -2.614741, -0.783807, 1.570796, 1.654510],accel_mss,speed_ms,0,blend_radius_m)
    |   movel([0.084029, -1.313805, -2.614764, -0.783821, 1.570796, 1.654826],accel_mss,speed_ms,0,blend_radius_m)
    |   movel([0.084275, -1.313954, -2.614672, -0.783763, 1.570796, 1.655071],accel_mss,speed_ms,0,blend_radius_m)
    |   movel([0.084281, -1.314246, -2.614492, -0.783650, 1.570796, 1.655077],accel_mss,speed_ms,0,blend_radius_m)
    |   movel([0.084076, -1.314711, -2.614206, -0.783471, 1.570796, 1.654872],accel_mss,speed_ms,0,blend_radius_m)
    |   movel([0.083648, -1.315836, -2.613514, -0.783039, 1.570796, 1.654444],accel_mss,speed_ms,0,blend_radius_m)
    |   movel([0.083205, -1.317019, -2.612783, -0.782587, 1.570796, 1.654001],accel_mss,speed_ms,0,blend_radius_m)
    |   movel([0.083202, -1.317302, -2.612608, -0.782479, 1.570796, 1.653998],accel_mss,speed_ms,0,blend_radius_m)
    |   movel([0.083652, -1.317193, -2.612675, -0.782520, 1.570796, 1.654448],accel_mss,speed_ms,0,blend_radius_m)
    |   movel([0.084222, -1.316970, -2.612813, -0.782605, 1.570796, 1.655019],accel_mss,speed_ms,0,blend_radius_m)
    |   movel([0.084649, -1.316806, -2.612915, -0.782668, 1.570796, 1.655445],accel_mss,speed_ms,0,blend_radius_m)
    |   movel([0.085028, -1.316673, -2.612997, -0.782719, 1.570796, 1.655825],accel_mss,speed_ms,0,blend_radius_m)
    |   movel([0.085344, -1.316573, -2.613059, -0.782757, 1.570796, 1.656140],accel_mss,speed_ms,0,blend_radius_m)
    |   movel([0.085547, -1.316717, -2.612970, -0.782702, 1.570796, 1.656343],accel_mss,speed_ms,0,blend_radius_m)
    |   movel([0.085460, -1.317124, -2.612719, -0.782547, 1.570796, 1.656257],accel_mss,speed_ms,0,blend_radius_m)
    |   movel([0.084802, -1.318680, -2.611754, -0.781955, 1.570796, 1.655598],accel_mss,speed_ms,0,blend_radius_m)
    |   movel([0.084057, -1.320391, -2.610691, -0.781307, 1.570796, 1.654853],accel_mss,speed_ms,0,blend_radius_m)
    |   movel([0.083277, -1.322119, -2.609613, -0.780657, 1.570796, 1.654073],accel_mss,speed_ms,0,blend_radius_m)
    |   movel([0.082971, -1.322793, -2.609192, -0.780405, 1.570796, 1.653767],accel_mss,speed_ms,0,blend_radius_m)
    |   movel([0.082683, -1.323437, -2.608788, -0.780164, 1.570796, 1.653479],accel_mss,speed_ms,0,blend_radius_m)
    |   movel([0.082444, -1.323982, -2.608446, -0.779961, 1.570796, 1.653241],accel_mss,speed_ms,0,blend_radius_m)
    |   movel([0.082332, -1.324263, -2.608270, -0.779856, 1.570796, 1.653129],accel_mss,speed_ms,0,blend_radius_m)
    |   movel([0.082154, -1.324637, -2.608035, -0.779717, 1.570796, 1.652950],accel_mss,speed_ms,0,blend_radius_m)
    |   movel([0.081915, -1.324973, -2.607824, -0.779592, 1.570796, 1.652711],accel_mss,speed_ms,0,blend_radius_m)
    |   movel([0.081676, -1.325197, -2.607683, -0.779509, 1.570796, 1.652472],accel_mss,speed_ms,0,blend_radius_m)
    |   speed_ms = 0.003
    |   movel([0.081492, -1.328688, -2.609225, -0.774476, 1.570796, 1.652288],accel_mss,speed_ms,0,blend_radius_m)
    |   speed_ms = 0.007
    |   movel([0.081341, -1.328466, -2.609366, -0.774557, 1.570796, 1.652138],accel_mss,speed_ms,0,blend_radius_m)
    |   movel([0.081467, -1.327621, -2.609900, -0.774869, 1.570796, 1.652263],accel_mss,speed_ms,0,blend_radius_m)
    |   movel([0.081769, -1.326371, -2.610687, -0.775331, 1.570796, 1.652565],accel_mss,speed_ms,0,blend_radius_m)
    |   movel([0.082314, -1.324569, -2.611819, -0.776001, 1.570796, 1.653110],accel_mss,speed_ms,0,blend_radius_m)
    |   movel([0.082603, -1.323582, -2.612437, -0.776370, 1.570796, 1.653400],accel_mss,speed_ms,0,blend_radius_m)
    |   movel([0.082660, -1.323095, -2.612741, -0.776553, 1.570796, 1.653456],accel_mss,speed_ms,0,blend_radius_m)
    |   movel([0.082527, -1.322934, -2.612842, -0.776613, 1.570796, 1.653323],accel_mss,speed_ms,0,blend_radius_m)
    |   movel([0.082236, -1.322994, -2.612804, -0.776590, 1.570796, 1.653033],accel_mss,speed_ms,0,blend_radius_m)
    |   movel([0.081751, -1.323241, -2.612650, -0.776498, 1.570796, 1.652547],accel_mss,speed_ms,0,blend_radius_m)
    |   movel([0.081384, -1.323420, -2.612538, -0.776431, 1.570796, 1.652181],accel_mss,speed_ms,0,blend_radius_m)
    |   movel([0.081002, -1.323604, -2.612423, -0.776362, 1.570796, 1.651798],accel_mss,speed_ms,0,blend_radius_m)
    |   movel([0.080195, -1.323913, -2.612230, -0.776246, 1.570796, 1.650992],accel_mss,speed_ms,0,blend_radius_m)
    |   movel([0.079870, -1.323817, -2.612290, -0.776282, 1.570796, 1.650667],accel_mss,speed_ms,0,blend_radius_m)
    |   movel([0.079791, -1.323313, -2.612605, -0.776471, 1.570796, 1.650588],accel_mss,speed_ms,0,blend_radius_m)
    |   movel([0.079966, -1.321386, -2.613807, -0.777196, 1.570796, 1.650762],accel_mss,speed_ms,0,blend_radius_m)
    |   movel([0.080077, -1.320375, -2.614436, -0.777578, 1.570796, 1.650873],accel_mss,speed_ms,0,blend_radius_m)
    |   movel([0.080182, -1.319602, -2.614916, -0.777871, 1.570796, 1.650979],accel_mss,speed_ms,0,blend_radius_m)
    |   movel([0.080285, -1.319004, -2.615287, -0.778098, 1.570796, 1.651081],accel_mss,speed_ms,0,blend_radius_m)
    |   movel([0.080559, -1.318652, -2.615504, -0.778232, 1.570796, 1.651355],accel_mss,speed_ms,0,blend_radius_m)
    |   movel([0.080916, -1.318448, -2.615631, -0.778310, 1.570796, 1.651713],accel_mss,speed_ms,0,blend_radius_m)
    |   movel([0.081474, -1.318181, -2.615796, -0.778412, 1.570796, 1.652271],accel_mss,speed_ms,0,blend_radius_m)
    |   movel([0.082380, -1.317797, -2.616034, -0.778559, 1.570796, 1.653176],accel_mss,speed_ms,0,blend_radius_m)
    |   movel([0.083212, -1.317464, -2.616239, -0.778686, 1.570796, 1.654008],accel_mss,speed_ms,0,blend_radius_m)
    |   movel([0.083713, -1.317304, -2.616338, -0.778747, 1.570796, 1.654510],accel_mss,speed_ms,0,blend_radius_m)
    |   movel([0.084029, -1.317267, -2.616361, -0.778761, 1.570796, 1.654826],accel_mss,speed_ms,0,blend_radius_m)
    |   movel([0.084275, -1.317416, -2.616269, -0.778704, 1.570796, 1.655071],accel_mss,speed_ms,0,blend_radius_m)
    |   movel([0.084281, -1.317708, -2.616088, -0.778593, 1.570796, 1.655077],accel_mss,speed_ms,0,blend_radius_m)
    |   movel([0.084076, -1.318171, -2.615802, -0.778416, 1.570796, 1.654872],accel_mss,speed_ms,0,blend_radius_m)
    |   movel([0.083648, -1.319294, -2.615107, -0.777988, 1.570796, 1.654444],accel_mss,speed_ms,0,blend_radius_m)
    |   movel([0.083205, -1.320474, -2.614375, -0.777540, 1.570796, 1.654001],accel_mss,speed_ms,0,blend_radius_m)
    |   movel([0.083202, -1.320756, -2.614200, -0.777434, 1.570796, 1.653998],accel_mss,speed_ms,0,blend_radius_m)
    |   movel([0.083652, -1.320648, -2.614267, -0.777475, 1.570796, 1.654448],accel_mss,speed_ms,0,blend_radius_m)
    |   movel([0.084222, -1.320425, -2.614405, -0.777559, 1.570796, 1.655019],accel_mss,speed_ms,0,blend_radius_m)
    |   movel([0.084649, -1.320261, -2.614507, -0.777621, 1.570796, 1.655445],accel_mss,speed_ms,0,blend_radius_m)
    |   movel([0.085028, -1.320129, -2.614589, -0.777671, 1.570796, 1.655825],accel_mss,speed_ms,0,blend_radius_m)
    |   movel([0.085344, -1.320029, -2.614651, -0.777709, 1.570796, 1.656140],accel_mss,speed_ms,0,blend_radius_m)
    |   movel([0.085547, -1.320173, -2.614562, -0.777654, 1.570796, 1.656343],accel_mss,speed_ms,0,blend_radius_m)
    |   movel([0.085460, -1.320578, -2.614310, -0.777501, 1.570796, 1.656257],accel_mss,speed_ms,0,blend_radius_m)
    |   movel([0.084802, -1.322131, -2.613343, -0.776915, 1.570796, 1.655598],accel_mss,speed_ms,0,blend_radius_m)
    |   movel([0.084057, -1.323838, -2.612277, -0.776274, 1.570796, 1.654853],accel_mss,speed_ms,0,blend_radius_m)
    |   movel([0.083277, -1.325561, -2.611196, -0.775632, 1.570796, 1.654073],accel_mss,speed_ms,0,blend_radius_m)
    |   movel([0.082971, -1.326234, -2.610773, -0.775382, 1.570796, 1.653767],accel_mss,speed_ms,0,blend_radius_m)
    |   movel([0.082683, -1.326877, -2.610369, -0.775144, 1.570796, 1.653479],accel_mss,speed_ms,0,blend_radius_m)
    |   movel([0.082444, -1.327420, -2.610026, -0.774943, 1.570796, 1.653241],accel_mss,speed_ms,0,blend_radius_m)
    |   movel([0.082332, -1.327700, -2.609849, -0.774839, 1.570796, 1.653129],accel_mss,speed_ms,0,blend_radius_m)
    |   movel([0.082154, -1.328074, -2.609613, -0.774702, 1.570796, 1.652950],accel_mss,speed_ms,0,blend_radius_m)
    |   movel([0.081915, -1.328409, -2.609402, -0.774578, 1.570796, 1.652711],accel_mss,speed_ms,0,blend_radius_m)
    |   movel([0.081676, -1.328633, -2.609260, -0.774496, 1.570796, 1.652472],accel_mss,speed_ms,0,blend_radius_m)
    |   speed_ms = 0.003
    |   movel([0.081492, -1.315103, -2.602865, -0.794421, 1.570796, 1.652288],accel_mss,speed_ms,0,blend_radius_m)
    |   speed_ms = 1.000
    |   movel([0.081492, -1.289170, -2.589753, -0.833466, 1.570796, 1.652288],accel_mss,speed_ms,0,blend_radius_m)
    |   movel([0.084778, -1.290377, -2.589031, -0.832981, 1.570796, 1.655574],accel_mss,speed_ms,0,blend_radius_m)
    |   movel([0.084778, -1.316292, -2.602127, -0.793970, 1.570796, 1.655574],accel_mss,speed_ms,0,blend_radius_m)
    |   speed_ms = 0.003
    |   movel([0.084778, -1.326433, -2.606904, -0.779052, 1.570796, 1.655574],accel_mss,speed_ms,0,blend_radius_m)
    |   speed_ms = 0.007
    |   movel([0.090842, -1.323774, -2.608577, -0.780038, 1.570796, 1.661638],accel_mss,speed_ms,0,blend_radius_m)
    |   movel([0.097024, -1.321322, -2.610111, -0.780956, 1.570796, 1.667820],accel_mss,speed_ms,0,blend_radius_m)
    |   movel([0.098922, -1.320620, -2.610549, -0.781221, 1.570796, 1.669718],accel_mss,speed_ms,0,blend_radius_m)
    |   movel([0.099688, -1.320397, -2.610687, -0.781305, 1.570796, 1.670484],accel_mss,speed_ms,0,blend_radius_m)
    |   movel([0.100116, -1.320391, -2.610691, -0.781307, 1.570796, 1.670912],accel_mss,speed_ms,0,blend_radius_m)
    |   movel([0.100432, -1.320571, -2.610579, -0.781239, 1.570796, 1.671229],accel_mss,speed_ms,0,blend_radius_m)
    |   movel([0.100558, -1.320745, -2.610471, -0.781174, 1.570796, 1.671354],accel_mss,speed_ms,0,blend_radius_m)
    |   movel([0.100527, -1.321057, -2.610276, -0.781056, 1.570796, 1.671323],accel_mss,speed_ms,0,blend_radius_m)
    |   movel([0.100222, -1.321346, -2.610096, -0.780947, 1.570796, 1.671018],accel_mss,speed_ms,0,blend_radius_m)
    |   movel([0.099520, -1.321694, -2.609879, -0.780817, 1.570796, 1.670316],accel_mss,speed_ms,0,blend_radius_m)
    |   movel([0.098688, -1.322091, -2.609630, -0.780668, 1.570796, 1.669485],accel_mss,speed_ms,0,blend_radius_m)
    |   movel([0.097742, -1.322527, -2.609358, -0.780504, 1.570796, 1.668538],accel_mss,speed_ms,0,blend_radius_m)
    |   movel([0.096707, -1.322998, -2.609063, -0.780328, 1.570796, 1.667503],accel_mss,speed_ms,0,blend_radius_m)
    |   movel([0.095604, -1.323499, -2.608749, -0.780141, 1.570796, 1.666400],accel_mss,speed_ms,0,blend_radius_m)
    |   movel([0.094597, -1.323965, -2.608457, -0.779967, 1.570796, 1.665393],accel_mss,speed_ms,0,blend_radius_m)
    |   movel([0.093881, -1.324296, -2.608249, -0.779844, 1.570796, 1.664677],accel_mss,speed_ms,0,blend_radius_m)
    |   movel([0.092978, -1.324716, -2.607985, -0.779688, 1.570796, 1.663774],accel_mss,speed_ms,0,blend_radius_m)
    |   movel([0.090797, -1.325723, -2.607352, -0.779314, 1.570796, 1.661593],accel_mss,speed_ms,0,blend_radius_m)
    |   movel([0.088204, -1.326921, -2.606596, -0.778872, 1.570796, 1.659000],accel_mss,speed_ms,0,blend_radius_m)
    |   movel([0.085405, -1.328216, -2.605777, -0.778396, 1.570796, 1.656201],accel_mss,speed_ms,0,blend_radius_m)
    |   movel([0.082317, -1.329650, -2.604868, -0.777871, 1.570796, 1.653113],accel_mss,speed_ms,0,blend_radius_m)
    |   movel([0.078847, -1.331268, -2.603839, -0.777282, 1.570796, 1.649643],accel_mss,speed_ms,0,blend_radius_m)
    |   movel([0.075532, -1.332819, -2.602849, -0.776722, 1.570796, 1.646329],accel_mss,speed_ms,0,blend_radius_m)
    |   movel([0.072957, -1.334028, -2.602074, -0.776286, 1.570796, 1.643754],accel_mss,speed_ms,0,blend_radius_m)
    |   movel([0.070326, -1.335262, -2.601283, -0.775845, 1.570796, 1.641122],accel_mss,speed_ms,0,blend_radius_m)
    |   movel([0.068708, -1.336000, -2.600808, -0.775581, 1.570796, 1.639505],accel_mss,speed_ms,0,blend_radius_m)
    |   movel([0.067572, -1.336501, -2.600485, -0.775403, 1.570796, 1.638368],accel_mss,speed_ms,0,blend_radius_m)
    |   movel([0.067250, -1.336369, -2.600570, -0.775450, 1.570796, 1.638047],accel_mss,speed_ms,0,blend_radius_m)
    |   movel([0.067250, -1.336102, -2.600742, -0.775545, 1.570796, 1.638047],accel_mss,speed_ms,0,blend_radius_m)
    |   movel([0.067376, -1.335776, -2.600952, -0.775661, 1.570796, 1.638173],accel_mss,speed_ms,0,blend_radius_m)
    |   movel([0.067604, -1.335465, -2.601152, -0.775772, 1.570796, 1.638401],accel_mss,speed_ms,0,blend_radius_m)
    |   movel([0.067983, -1.335141, -2.601360, -0.775888, 1.570796, 1.638779],accel_mss,speed_ms,0,blend_radius_m)
    |   movel([0.068669, -1.334712, -2.601636, -0.776041, 1.570796, 1.639465],accel_mss,speed_ms,0,blend_radius_m)
    |   movel([0.069880, -1.334026, -2.602076, -0.776287, 1.570796, 1.640676],accel_mss,speed_ms,0,blend_radius_m)
    |   movel([0.072622, -1.332531, -2.603033, -0.776825, 1.570796, 1.643418],accel_mss,speed_ms,0,blend_radius_m)
    |   movel([0.078735, -1.329339, -2.605065, -0.777984, 1.570796, 1.649532],accel_mss,speed_ms,0,blend_radius_m)
    |   movel([0.084778, -1.326433, -2.606904, -0.779052, 1.570796, 1.655574],accel_mss,speed_ms,0,blend_radius_m)
    |   speed_ms = 0.003
    |   movel([0.084778, -1.329866, -2.608480, -0.774044, 1.570796, 1.655574],accel_mss,speed_ms,0,blend_radius_m)
    |   speed_ms = 0.007
    |   movel([0.090842, -1.327213, -2.610157, -0.775019, 1.570796, 1.661638],accel_mss,speed_ms,0,blend_radius_m)
    |   movel([0.097024, -1.324766, -2.611695, -0.775928, 1.570796, 1.667820],accel_mss,speed_ms,0,blend_radius_m)
    |   movel([0.098922, -1.324066, -2.612134, -0.776189, 1.570796, 1.669718],accel_mss,speed_ms,0,blend_radius_m)
    |   movel([0.099688, -1.323844, -2.612273, -0.776272, 1.570796, 1.670484],accel_mss,speed_ms,0,blend_radius_m)
    |   movel([0.100116, -1.323838, -2.612277, -0.776274, 1.570796, 1.670912],accel_mss,speed_ms,0,blend_radius_m)
    |   movel([0.100432, -1.324018, -2.612164, -0.776207, 1.570796, 1.671229],accel_mss,speed_ms,0,blend_radius_m)
    |   movel([0.100558, -1.324191, -2.612056, -0.776142, 1.570796, 1.671354],accel_mss,speed_ms,0,blend_radius_m)
    |   movel([0.100527, -1.324503, -2.611860, -0.776026, 1.570796, 1.671323],accel_mss,speed_ms,0,blend_radius_m)
    |   movel([0.100222, -1.324790, -2.611680, -0.775919, 1.570796, 1.671018],accel_mss,speed_ms,0,blend_radius_m)
    |   movel([0.099520, -1.325137, -2.611462, -0.775789, 1.570796, 1.670316],accel_mss,speed_ms,0,blend_radius_m)
    |   movel([0.098688, -1.325534, -2.611213, -0.775642, 1.570796, 1.669485],accel_mss,speed_ms,0,blend_radius_m)
    |   movel([0.097742, -1.325969, -2.610940, -0.775480, 1.570796, 1.668538],accel_mss,speed_ms,0,blend_radius_m)
    |   movel([0.096707, -1.326438, -2.610645, -0.775306, 1.570796, 1.667503],accel_mss,speed_ms,0,blend_radius_m)
    |   movel([0.095604, -1.326939, -2.610330, -0.775121, 1.570796, 1.666400],accel_mss,speed_ms,0,blend_radius_m)
    |   movel([0.094597, -1.327403, -2.610037, -0.774949, 1.570796, 1.665393],accel_mss,speed_ms,0,blend_radius_m)
    |   movel([0.093881, -1.327733, -2.609828, -0.774827, 1.570796, 1.664677],accel_mss,speed_ms,0,blend_radius_m)
    |   movel([0.092978, -1.328152, -2.609564, -0.774673, 1.570796, 1.663774],accel_mss,speed_ms,0,blend_radius_m)
    |   movel([0.090797, -1.329157, -2.608929, -0.774303, 1.570796, 1.661593],accel_mss,speed_ms,0,blend_radius_m)
    |   movel([0.088204, -1.330352, -2.608171, -0.773866, 1.570796, 1.659000],accel_mss,speed_ms,0,blend_radius_m)
    |   movel([0.085405, -1.331644, -2.607350, -0.773395, 1.570796, 1.656201],accel_mss,speed_ms,0,blend_radius_m)
    |   movel([0.082317, -1.333074, -2.606438, -0.772876, 1.570796, 1.653113],accel_mss,speed_ms,0,blend_radius_m)
    |   movel([0.078847, -1.334688, -2.605406, -0.772294, 1.570796, 1.649643],accel_mss,speed_ms,0,blend_radius_m)
    |   movel([0.075532, -1.336235, -2.604414, -0.771740, 1.570796, 1.646329],accel_mss,speed_ms,0,blend_radius_m)
    |   movel([0.072957, -1.337442, -2.603637, -0.771310, 1.570796, 1.643754],accel_mss,speed_ms,0,blend_radius_m)
    |   movel([0.070326, -1.338672, -2.602844, -0.770873, 1.570796, 1.641122],accel_mss,speed_ms,0,blend_radius_m)
    |   movel([0.068708, -1.339409, -2.602367, -0.770613, 1.570796, 1.639505],accel_mss,speed_ms,0,blend_radius_m)
    |   movel([0.067572, -1.339908, -2.602044, -0.770437, 1.570796, 1.638368],accel_mss,speed_ms,0,blend_radius_m)
    |   movel([0.067250, -1.339777, -2.602129, -0.770483, 1.570796, 1.638047],accel_mss,speed_ms,0,blend_radius_m)
    |   movel([0.067250, -1.339511, -2.602301, -0.770577, 1.570796, 1.638047],accel_mss,speed_ms,0,blend_radius_m)
    |   movel([0.067376, -1.339185, -2.602512, -0.770692, 1.570796, 1.638173],accel_mss,speed_ms,0,blend_radius_m)
    |   movel([0.067604, -1.338875, -2.602713, -0.770802, 1.570796, 1.638401],accel_mss,speed_ms,0,blend_radius_m)
    |   movel([0.067983, -1.338552, -2.602921, -0.770916, 1.570796, 1.638779],accel_mss,speed_ms,0,blend_radius_m)
    |   movel([0.068669, -1.338124, -2.603197, -0.771067, 1.570796, 1.639465],accel_mss,speed_ms,0,blend_radius_m)
    |   movel([0.069880, -1.337439, -2.603639, -0.771311, 1.570796, 1.640676],accel_mss,speed_ms,0,blend_radius_m)
    |   movel([0.072622, -1.335949, -2.604598, -0.771843, 1.570796, 1.643418],accel_mss,speed_ms,0,blend_radius_m)
    |   movel([0.078735, -1.332764, -2.606636, -0.772988, 1.570796, 1.649532],accel_mss,speed_ms,0,blend_radius_m)
    |   movel([0.084778, -1.329866, -2.608480, -0.774044, 1.570796, 1.655574],accel_mss,speed_ms,0,blend_radius_m)
    |   speed_ms = 0.003
    |   movel([0.084778, -1.316292, -2.602127, -0.793970, 1.570796, 1.655574],accel_mss,speed_ms,0,blend_radius_m)
    |   speed_ms = 1.000
    |   movel([0.084778, -1.290377, -2.589031, -0.832981, 1.570796, 1.655574],accel_mss,speed_ms,0,blend_radius_m)
    |   movel([0.084148, -1.290304, -2.589074, -0.833010, 1.570796, 1.654945],accel_mss,speed_ms,0,blend_radius_m)
    |   movel([0.084148, -1.316221, -2.602171, -0.793997, 1.570796, 1.654945],accel_mss,speed_ms,0,blend_radius_m)
    |   speed_ms = 0.003
    |   movel([0.084148, -1.326362, -2.606949, -0.779078, 1.570796, 1.654945],accel_mss,speed_ms,0,blend_radius_m)
    |   speed_ms = 0.007
    |   movel([0.080371, -1.328162, -2.605812, -0.778416, 1.570796, 1.651168],accel_mss,speed_ms,0,blend_radius_m)
    |   movel([0.077408, -1.329664, -2.604859, -0.777866, 1.570796, 1.648205],accel_mss,speed_ms,0,blend_radius_m)
    |   movel([0.073168, -1.331900, -2.603435, -0.777053, 1.570796, 1.643964],accel_mss,speed_ms,0,blend_radius_m)
    |   movel([0.068676, -1.334302, -2.601899, -0.776188, 1.570796, 1.639472],accel_mss,speed_ms,0,blend_radius_m)
    |   movel([0.068123, -1.334676, -2.601659, -0.776054, 1.570796, 1.638919],accel_mss,speed_ms,0,blend_radius_m)
    |   movel([0.067836, -1.334677, -2.601658, -0.776054, 1.570796, 1.638633],accel_mss,speed_ms,0,blend_radius_m)
    |   movel([0.067589, -1.333691, -2.602291, -0.776408, 1.570796, 1.638385],accel_mss,speed_ms,0,blend_radius_m)
    |   movel([0.067346, -1.332066, -2.603330, -0.776993, 1.570796, 1.638142],accel_mss,speed_ms,0,blend_radius_m)
    |   movel([0.067096, -1.329414, -2.605018, -0.777957, 1.570796, 1.637892],accel_mss,speed_ms,0,blend_radius_m)
    |   movel([0.067029, -1.326857, -2.606636, -0.778895, 1.570796, 1.637826],accel_mss,speed_ms,0,blend_radius_m)
    |   movel([0.067221, -1.323815, -2.608551, -0.780023, 1.570796, 1.638017],accel_mss,speed_ms,0,blend_radius_m)
    |   movel([0.067565, -1.320910, -2.610368, -0.781111, 1.570796, 1.638361],accel_mss,speed_ms,0,blend_radius_m)
    |   movel([0.068023, -1.319911, -2.610990, -0.781488, 1.570796, 1.638820],accel_mss,speed_ms,0,blend_radius_m)
    |   movel([0.068550, -1.319416, -2.611298, -0.781676, 1.570796, 1.639347],accel_mss,speed_ms,0,blend_radius_m)
    |   movel([0.070937, -1.317784, -2.612310, -0.782295, 1.570796, 1.641733],accel_mss,speed_ms,0,blend_radius_m)
    |   movel([0.073484, -1.316103, -2.613349, -0.782937, 1.570796, 1.644281],accel_mss,speed_ms,0,blend_radius_m)
    |   movel([0.075813, -1.314653, -2.614242, -0.783494, 1.570796, 1.646609],accel_mss,speed_ms,0,blend_radius_m)
    |   movel([0.078779, -1.312938, -2.615295, -0.784156, 1.570796, 1.649576],accel_mss,speed_ms,0,blend_radius_m)
    |   movel([0.081413, -1.311574, -2.616130, -0.784685, 1.570796, 1.652209],accel_mss,speed_ms,0,blend_radius_m)
    |   movel([0.084118, -1.310360, -2.616871, -0.785158, 1.570796, 1.654915],accel_mss,speed_ms,0,blend_radius_m)
    |   movel([0.087305, -1.309106, -2.617634, -0.785649, 1.570796, 1.658101],accel_mss,speed_ms,0,blend_radius_m)
    |   movel([0.089778, -1.308243, -2.618158, -0.785988, 1.570796, 1.660575],accel_mss,speed_ms,0,blend_radius_m)
    |   movel([0.092672, -1.307345, -2.618702, -0.786342, 1.570796, 1.663468],accel_mss,speed_ms,0,blend_radius_m)
    |   movel([0.095427, -1.306558, -2.619178, -0.786653, 1.570796, 1.666223],accel_mss,speed_ms,0,blend_radius_m)
    |   movel([0.096203, -1.306481, -2.619225, -0.786683, 1.570796, 1.666999],accel_mss,speed_ms,0,blend_radius_m)
    |   movel([0.096612, -1.306789, -2.619039, -0.786561, 1.570796, 1.667408],accel_mss,speed_ms,0,blend_radius_m)
    |   movel([0.096874, -1.307161, -2.618814, -0.786415, 1.570796, 1.667670],accel_mss,speed_ms,0,blend_radius_m)
    |   movel([0.097202, -1.307715, -2.618478, -0.786196, 1.570796, 1.667998],accel_mss,speed_ms,0,blend_radius_m)
    |   movel([0.098014, -1.309498, -2.617396, -0.785496, 1.570796, 1.668810],accel_mss,speed_ms,0,blend_radius_m)
    |   movel([0.098672, -1.311674, -2.616069, -0.784646, 1.570796, 1.669469],accel_mss,speed_ms,0,blend_radius_m)
    |   movel([0.099188, -1.314269, -2.614478, -0.783642, 1.570796, 1.669984],accel_mss,speed_ms,0,blend_radius_m)
    |   movel([0.099569, -1.317326, -2.612593, -0.782470, 1.570796, 1.670365],accel_mss,speed_ms,0,blend_radius_m)
    |   movel([0.099684, -1.318625, -2.611789, -0.781975, 1.570796, 1.670481],accel_mss,speed_ms,0,blend_radius_m)
    |   movel([0.099703, -1.319328, -2.611352, -0.781709, 1.570796, 1.670499],accel_mss,speed_ms,0,blend_radius_m)
    |   movel([0.099661, -1.319764, -2.611081, -0.781544, 1.570796, 1.670458],accel_mss,speed_ms,0,blend_radius_m)
    |   movel([0.099398, -1.320054, -2.610901, -0.781434, 1.570796, 1.670194],accel_mss,speed_ms,0,blend_radius_m)
    |   movel([0.098670, -1.320347, -2.610718, -0.781324, 1.570796, 1.669466],accel_mss,speed_ms,0,blend_radius_m)
    |   movel([0.097818, -1.320681, -2.610510, -0.781198, 1.570796, 1.668615],accel_mss,speed_ms,0,blend_radius_m)
    |   movel([0.096841, -1.321053, -2.610278, -0.781057, 1.570796, 1.667638],accel_mss,speed_ms,0,blend_radius_m)
    |   movel([0.092668, -1.322683, -2.609260, -0.780446, 1.570796, 1.663465],accel_mss,speed_ms,0,blend_radius_m)
    |   movel([0.088344, -1.324493, -2.608126, -0.779771, 1.570796, 1.659140],accel_mss,speed_ms,0,blend_radius_m)
    |   movel([0.084148, -1.326362, -2.606949, -0.779078, 1.570796, 1.654945],accel_mss,speed_ms,0,blend_radius_m)
    |   speed_ms = 0.003
    |   movel([0.084148, -1.329795, -2.608525, -0.774070, 1.570796, 1.654945],accel_mss,speed_ms,0,blend_radius_m)
    |   speed_ms = 0.007
    |   movel([0.080371, -1.331590, -2.607385, -0.773415, 1.570796, 1.651168],accel_mss,speed_ms,0,blend_radius_m)
    |   movel([0.077408, -1.333089, -2.606429, -0.772871, 1.570796, 1.648205],accel_mss,speed_ms,0,blend_radius_m)
    |   movel([0.073168, -1.335319, -2.605002, -0.772068, 1.570796, 1.643964],accel_mss,speed_ms,0,blend_radius_m)
    |   movel([0.068676, -1.337715, -2.603461, -0.771213, 1.570796, 1.639472],accel_mss,speed_ms,0,blend_radius_m)
    |   movel([0.068123, -1.338088, -2.603221, -0.771080, 1.570796, 1.638919],accel_mss,speed_ms,0,blend_radius_m)
    |   movel([0.067836, -1.338089, -2.603220, -0.771080, 1.570796, 1.638633],accel_mss,speed_ms,0,blend_radius_m)
    |   movel([0.067589, -1.337105, -2.603854, -0.771430, 1.570796, 1.638385],accel_mss,speed_ms,0,blend_radius_m)
    |   movel([0.067346, -1.335484, -2.604896, -0.772009, 1.570796, 1.638142],accel_mss,speed_ms,0,blend_radius_m)
    |   movel([0.067096, -1.332839, -2.606589, -0.772962, 1.570796, 1.637892],accel_mss,speed_ms,0,blend_radius_m)
    |   movel([0.067029, -1.330288, -2.608211, -0.773889, 1.570796, 1.637826],accel_mss,speed_ms,0,blend_radius_m)
    |   movel([0.067221, -1.327253, -2.610131, -0.775004, 1.570796, 1.638017],accel_mss,speed_ms,0,blend_radius_m)
    |   movel([0.067565, -1.324356, -2.611953, -0.776081, 1.570796, 1.638361],accel_mss,speed_ms,0,blend_radius_m)
    |   movel([0.068023, -1.323359, -2.612577, -0.776454, 1.570796, 1.638820],accel_mss,speed_ms,0,blend_radius_m)
    |   movel([0.068550, -1.322865, -2.612885, -0.776639, 1.570796, 1.639347],accel_mss,speed_ms,0,blend_radius_m)
    |   movel([0.070937, -1.321237, -2.613900, -0.777252, 1.570796, 1.641733],accel_mss,speed_ms,0,blend_radius_m)
    |   movel([0.073484, -1.319560, -2.614942, -0.777887, 1.570796, 1.644281],accel_mss,speed_ms,0,blend_radius_m)
    |   movel([0.075813, -1.318113, -2.615838, -0.778438, 1.570796, 1.646609],accel_mss,speed_ms,0,blend_radius_m)
    |   movel([0.078779, -1.316403, -2.616894, -0.779093, 1.570796, 1.649576],accel_mss,speed_ms,0,blend_radius_m)
    |   movel([0.081413, -1.315042, -2.617730, -0.779617, 1.570796, 1.652209],accel_mss,speed_ms,0,blend_radius_m)
    |   movel([0.084118, -1.313831, -2.618473, -0.780085, 1.570796, 1.654915],accel_mss,speed_ms,0,blend_radius_m)
    |   movel([0.087305, -1.312579, -2.619239, -0.780571, 1.570796, 1.658101],accel_mss,speed_ms,0,blend_radius_m)
    |   movel([0.089778, -1.311718, -2.619764, -0.780906, 1.570796, 1.660575],accel_mss,speed_ms,0,blend_radius_m)
    |   movel([0.092672, -1.310823, -2.620310, -0.781256, 1.570796, 1.663468],accel_mss,speed_ms,0,blend_radius_m)
    |   movel([0.095427, -1.310038, -2.620787, -0.781564, 1.570796, 1.666223],accel_mss,speed_ms,0,blend_radius_m)
    |   movel([0.096203, -1.309960, -2.620834, -0.781594, 1.570796, 1.666999],accel_mss,speed_ms,0,blend_radius_m)
    |   movel([0.096612, -1.310268, -2.620648, -0.781474, 1.570796, 1.667408],accel_mss,speed_ms,0,blend_radius_m)
    |   movel([0.096874, -1.310638, -2.620422, -0.781328, 1.570796, 1.667670],accel_mss,speed_ms,0,blend_radius_m)
    |   movel([0.097202, -1.311192, -2.620085, -0.781112, 1.570796, 1.667998],accel_mss,speed_ms,0,blend_radius_m)
    |   movel([0.098014, -1.312970, -2.619000, -0.780419, 1.570796, 1.668810],accel_mss,speed_ms,0,blend_radius_m)
    |   movel([0.098672, -1.315142, -2.617669, -0.779578, 1.570796, 1.669469],accel_mss,speed_ms,0,blend_radius_m)
    |   movel([0.099188, -1.317731, -2.616074, -0.778584, 1.570796, 1.669984],accel_mss,speed_ms,0,blend_radius_m)
    |   movel([0.099569, -1.320780, -2.614184, -0.777424, 1.570796, 1.670365],accel_mss,speed_ms,0,blend_radius_m)
    |   movel([0.099684, -1.322076, -2.613377, -0.776935, 1.570796, 1.670481],accel_mss,speed_ms,0,blend_radius_m)
    |   movel([0.099703, -1.322777, -2.612940, -0.776672, 1.570796, 1.670499],accel_mss,speed_ms,0,blend_radius_m)
    |   movel([0.099661, -1.323212, -2.612668, -0.776509, 1.570796, 1.670458],accel_mss,speed_ms,0,blend_radius_m)
    |   movel([0.099398, -1.323501, -2.612487, -0.776400, 1.570796, 1.670194],accel_mss,speed_ms,0,blend_radius_m)
    |   movel([0.098670, -1.323794, -2.612304, -0.776291, 1.570796, 1.669466],accel_mss,speed_ms,0,blend_radius_m)
    |   movel([0.097818, -1.324127, -2.612096, -0.776166, 1.570796, 1.668615],accel_mss,speed_ms,0,blend_radius_m)
    |   movel([0.096841, -1.324498, -2.611863, -0.776027, 1.570796, 1.667638],accel_mss,speed_ms,0,blend_radius_m)
    |   movel([0.092668, -1.326124, -2.610842, -0.775423, 1.570796, 1.663465],accel_mss,speed_ms,0,blend_radius_m)
    |   movel([0.088344, -1.327930, -2.609704, -0.774755, 1.570796, 1.659140],accel_mss,speed_ms,0,blend_radius_m)
    |   movel([0.084148, -1.329795, -2.608525, -0.774070, 1.570796, 1.654945],accel_mss,speed_ms,0,blend_radius_m)
    |   speed_ms = 0.003
    |   movel([0.084148, -1.316221, -2.602171, -0.793997, 1.570796, 1.654945],accel_mss,speed_ms,0,blend_radius_m)
    |   speed_ms = 1.000
    |   movel([0.084148, -1.290304, -2.589074, -0.833010, 1.570796, 1.654945],accel_mss,speed_ms,0,blend_radius_m)
    |   movel([0.103618, -1.282197, -2.593889, -0.836303, 1.570796, 1.674414],accel_mss,speed_ms,0,blend_radius_m)
    |   movel([0.103618, -1.308235, -2.607092, -0.797062, 1.570796, 1.674414],accel_mss,speed_ms,0,blend_radius_m)
    |   speed_ms = 0.003
    |   movel([0.103618, -1.318431, -2.611909, -0.782049, 1.570796, 1.674414],accel_mss,speed_ms,0,blend_radius_m)
    |   speed_ms = 0.007
    |   movel([0.103637, -1.318157, -2.612079, -0.782153, 1.570796, 1.674433],accel_mss,speed_ms,0,blend_radius_m)
    |   movel([0.103885, -1.317021, -2.612782, -0.782586, 1.570796, 1.674681],accel_mss,speed_ms,0,blend_radius_m)
    |   movel([0.104417, -1.315534, -2.613700, -0.783155, 1.570796, 1.675214],accel_mss,speed_ms,0,blend_radius_m)
    |   movel([0.105039, -1.314112, -2.614575, -0.783702, 1.570796, 1.675836],accel_mss,speed_ms,0,blend_radius_m)
    |   movel([0.105483, -1.313585, -2.614898, -0.783906, 1.570796, 1.676279],accel_mss,speed_ms,0,blend_radius_m)
    |   movel([0.105791, -1.313406, -2.615008, -0.783975, 1.570796, 1.676587],accel_mss,speed_ms,0,blend_radius_m)
    |   movel([0.106222, -1.313247, -2.615105, -0.784036, 1.570796, 1.677018],accel_mss,speed_ms,0,blend_radius_m)
    |   movel([0.106665, -1.313136, -2.615174, -0.784079, 1.570796, 1.677462],accel_mss,speed_ms,0,blend_radius_m)
    |   movel([0.107028, -1.313106, -2.615192, -0.784091, 1.570796, 1.677825],accel_mss,speed_ms,0,blend_radius_m)
    |   movel([0.107242, -1.313211, -2.615128, -0.784050, 1.570796, 1.678039],accel_mss,speed_ms,0,blend_radius_m)
    |   movel([0.107306, -1.313480, -2.614963, -0.783946, 1.570796, 1.678102],accel_mss,speed_ms,0,blend_radius_m)
    |   movel([0.107218, -1.314076, -2.614597, -0.783716, 1.570796, 1.678014],accel_mss,speed_ms,0,blend_radius_m)
    |   movel([0.106840, -1.315758, -2.613562, -0.783069, 1.570796, 1.677636],accel_mss,speed_ms,0,blend_radius_m)
    |   movel([0.106420, -1.317549, -2.612455, -0.782385, 1.570796, 1.677217],accel_mss,speed_ms,0,blend_radius_m)
    |   movel([0.106260, -1.318107, -2.612110, -0.782172, 1.570796, 1.677056],accel_mss,speed_ms,0,blend_radius_m)
    |   movel([0.106100, -1.318394, -2.611932, -0.782063, 1.570796, 1.676897],accel_mss,speed_ms,0,blend_radius_m)
    |   movel([0.105428, -1.318749, -2.611711, -0.781928, 1.570796, 1.676224],accel_mss,speed_ms,0,blend_radius_m)
    |   movel([0.104756, -1.318864, -2.611640, -0.781885, 1.570796, 1.675553],accel_mss,speed_ms,0,blend_radius_m)
    |   movel([0.104107, -1.318923, -2.611604, -0.781862, 1.570796, 1.674903],accel_mss,speed_ms,0,blend_radius_m)
    |   movel([0.103793, -1.318857, -2.611645, -0.781887, 1.570796, 1.674589],accel_mss,speed_ms,0,blend_radius_m)
    |   movel([0.103635, -1.318631, -2.611785, -0.781973, 1.570796, 1.674432],accel_mss,speed_ms,0,blend_radius_m)
    |   speed_ms = 0.003
    |   movel([0.103618, -1.321882, -2.613498, -0.777009, 1.570796, 1.674414],accel_mss,speed_ms,0,blend_radius_m)
    |   speed_ms = 0.007
    |   movel([0.103637, -1.321609, -2.613669, -0.777111, 1.570796, 1.674433],accel_mss,speed_ms,0,blend_radius_m)
    |   movel([0.103885, -1.320476, -2.614373, -0.777540, 1.570796, 1.674681],accel_mss,speed_ms,0,blend_radius_m)
    |   movel([0.104417, -1.318992, -2.615294, -0.778103, 1.570796, 1.675214],accel_mss,speed_ms,0,blend_radius_m)
    |   movel([0.105039, -1.317574, -2.616171, -0.778644, 1.570796, 1.675836],accel_mss,speed_ms,0,blend_radius_m)
    |   movel([0.105483, -1.317048, -2.616496, -0.778845, 1.570796, 1.676279],accel_mss,speed_ms,0,blend_radius_m)
    |   movel([0.105791, -1.316870, -2.616606, -0.778914, 1.570796, 1.676587],accel_mss,speed_ms,0,blend_radius_m)
    |   movel([0.106222, -1.316711, -2.616703, -0.778974, 1.570796, 1.677018],accel_mss,speed_ms,0,blend_radius_m)
    |   movel([0.106665, -1.316600, -2.616772, -0.779017, 1.570796, 1.677462],accel_mss,speed_ms,0,blend_radius_m)
    |   movel([0.107028, -1.316570, -2.616790, -0.779028, 1.570796, 1.677825],accel_mss,speed_ms,0,blend_radius_m)
    |   movel([0.107242, -1.316675, -2.616726, -0.778988, 1.570796, 1.678039],accel_mss,speed_ms,0,blend_radius_m)
    |   movel([0.107306, -1.316943, -2.616561, -0.778886, 1.570796, 1.678102],accel_mss,speed_ms,0,blend_radius_m)
    |   movel([0.107218, -1.317538, -2.616193, -0.778658, 1.570796, 1.678014],accel_mss,speed_ms,0,blend_radius_m)
    |   movel([0.106840, -1.319216, -2.615155, -0.778018, 1.570796, 1.677636],accel_mss,speed_ms,0,blend_radius_m)
    |   movel([0.106420, -1.321002, -2.614046, -0.777340, 1.570796, 1.677217],accel_mss,speed_ms,0,blend_radius_m)
    |   movel([0.106260, -1.321559, -2.613699, -0.777130, 1.570796, 1.677056],accel_mss,speed_ms,0,blend_radius_m)
    |   movel([0.106100, -1.321846, -2.613521, -0.777022, 1.570796, 1.676897],accel_mss,speed_ms,0,blend_radius_m)
    |   movel([0.105428, -1.322200, -2.613300, -0.776889, 1.570796, 1.676224],accel_mss,speed_ms,0,blend_radius_m)
    |   movel([0.104756, -1.322315, -2.613228, -0.776846, 1.570796, 1.675553],accel_mss,speed_ms,0,blend_radius_m)
    |   movel([0.104107, -1.322373, -2.613192, -0.776824, 1.570796, 1.674903],accel_mss,speed_ms,0,blend_radius_m)
    |   movel([0.103793, -1.322308, -2.613233, -0.776848, 1.570796, 1.674589],accel_mss,speed_ms,0,blend_radius_m)
    |   movel([0.103635, -1.322082, -2.613374, -0.776933, 1.570796, 1.674432],accel_mss,speed_ms,0,blend_radius_m)
    |   speed_ms = 0.003
    |   movel([0.103618, -1.308235, -2.607092, -0.797062, 1.570796, 1.674414],accel_mss,speed_ms,0,blend_radius_m)
    |   speed_ms = 1.000
    |   movel([0.103618, -1.282197, -2.593889, -0.836303, 1.570796, 1.674414],accel_mss,speed_ms,0,blend_radius_m)
    |   movel([0.103813, -1.270306, -2.600804, -0.841279, 1.570796, 1.674610],accel_mss,speed_ms,0,blend_radius_m)
    |   movel([0.103813, -1.296516, -2.614163, -0.801711, 1.570796, 1.674610],accel_mss,speed_ms,0,blend_radius_m)
    |   speed_ms = 0.003
    |   movel([0.103813, -1.306788, -2.619039, -0.786562, 1.570796, 1.674610],accel_mss,speed_ms,0,blend_radius_m)
    |   speed_ms = 0.007
    |   movel([0.103818, -1.306456, -2.619240, -0.786693, 1.570796, 1.674615],accel_mss,speed_ms,0,blend_radius_m)
    |   movel([0.104142, -1.305715, -2.619687, -0.786987, 1.570796, 1.674938],accel_mss,speed_ms,0,blend_radius_m)
    |   movel([0.105377, -1.303033, -2.621301, -0.788055, 1.570796, 1.676173],accel_mss,speed_ms,0,blend_radius_m)
    |   movel([0.105952, -1.301774, -2.622055, -0.788560, 1.570796, 1.676748],accel_mss,speed_ms,0,blend_radius_m)
    |   movel([0.106444, -1.300670, -2.622715, -0.789004, 1.570796, 1.677240],accel_mss,speed_ms,0,blend_radius_m)
    |   movel([0.106854, -1.299726, -2.623277, -0.789385, 1.570796, 1.677650],accel_mss,speed_ms,0,blend_radius_m)
    |   movel([0.106834, -1.299363, -2.623494, -0.789532, 1.570796, 1.677630],accel_mss,speed_ms,0,blend_radius_m)
    |   movel([0.106601, -1.299322, -2.623518, -0.789549, 1.570796, 1.677397],accel_mss,speed_ms,0,blend_radius_m)
    |   movel([0.106084, -1.299434, -2.623451, -0.789504, 1.570796, 1.676881],accel_mss,speed_ms,0,blend_radius_m)
    |   movel([0.104894, -1.299801, -2.623233, -0.789355, 1.570796, 1.675691],accel_mss,speed_ms,0,blend_radius_m)
    |   movel([0.104141, -1.300033, -2.623094, -0.789261, 1.570796, 1.674938],accel_mss,speed_ms,0,blend_radius_m)
    |   movel([0.103630, -1.300168, -2.623014, -0.789207, 1.570796, 1.674427],accel_mss,speed_ms,0,blend_radius_m)
    |   movel([0.103281, -1.300238, -2.622973, -0.789179, 1.570796, 1.674077],accel_mss,speed_ms,0,blend_radius_m)
    |   movel([0.103139, -1.300064, -2.623076, -0.789249, 1.570796, 1.673936],accel_mss,speed_ms,0,blend_radius_m)
    |   movel([0.103501, -1.299189, -2.623597, -0.789603, 1.570796, 1.674298],accel_mss,speed_ms,0,blend_radius_m)
    |   movel([0.104030, -1.297983, -2.624314, -0.790092, 1.570796, 1.674826],accel_mss,speed_ms,0,blend_radius_m)
    |   movel([0.104855, -1.296189, -2.625376, -0.790824, 1.570796, 1.675651],accel_mss,speed_ms,0,blend_radius_m)
    |   movel([0.105571, -1.294665, -2.626275, -0.791449, 1.570796, 1.676367],accel_mss,speed_ms,0,blend_radius_m)
    |   movel([0.106206, -1.293339, -2.627055, -0.791995, 1.570796, 1.677002],accel_mss,speed_ms,0,blend_radius_m)
    |   movel([0.106762, -1.292196, -2.627726, -0.792467, 1.570796, 1.677558],accel_mss,speed_ms,0,blend_radius_m)
    |   movel([0.107086, -1.291849, -2.627929, -0.792611, 1.570796, 1.677883],accel_mss,speed_ms,0,blend_radius_m)
    |   movel([0.107542, -1.291653, -2.628044, -0.792692, 1.570796, 1.678339],accel_mss,speed_ms,0,blend_radius_m)
    |   movel([0.108293, -1.291386, -2.628200, -0.792803, 1.570796, 1.679089],accel_mss,speed_ms,0,blend_radius_m)
    |   movel([0.109705, -1.290927, -2.628468, -0.792993, 1.570796, 1.680502],accel_mss,speed_ms,0,blend_radius_m)
    |   movel([0.110994, -1.290524, -2.628704, -0.793161, 1.570796, 1.681790],accel_mss,speed_ms,0,blend_radius_m)
    |   movel([0.111769, -1.290303, -2.628832, -0.793253, 1.570796, 1.682565],accel_mss,speed_ms,0,blend_radius_m)
    |   movel([0.112276, -1.290181, -2.628904, -0.793304, 1.570796, 1.683072],accel_mss,speed_ms,0,blend_radius_m)
    |   movel([0.111888, -1.291179, -2.628321, -0.792889, 1.570796, 1.682685],accel_mss,speed_ms,0,blend_radius_m)
    |   movel([0.111324, -1.292151, -2.627752, -0.792486, 1.570796, 1.682120],accel_mss,speed_ms,0,blend_radius_m)
    |   movel([0.110646, -1.293277, -2.627092, -0.792020, 1.570796, 1.681442],accel_mss,speed_ms,0,blend_radius_m)
    |   movel([0.109696, -1.294842, -2.626171, -0.791376, 1.570796, 1.680492],accel_mss,speed_ms,0,blend_radius_m)
    |   movel([0.109237, -1.295653, -2.625692, -0.791043, 1.570796, 1.680034],accel_mss,speed_ms,0,blend_radius_m)
    |   movel([0.109006, -1.296136, -2.625407, -0.790845, 1.570796, 1.679802],accel_mss,speed_ms,0,blend_radius_m)
    |   movel([0.109167, -1.296352, -2.625280, -0.790757, 1.570796, 1.679964],accel_mss,speed_ms,0,blend_radius_m)
    |   movel([0.109462, -1.296309, -2.625305, -0.790775, 1.570796, 1.680258],accel_mss,speed_ms,0,blend_radius_m)
    |   movel([0.109933, -1.296190, -2.625375, -0.790823, 1.570796, 1.680729],accel_mss,speed_ms,0,blend_radius_m)
    |   movel([0.110719, -1.295949, -2.625518, -0.790922, 1.570796, 1.681516],accel_mss,speed_ms,0,blend_radius_m)
    |   movel([0.111646, -1.295667, -2.625685, -0.791038, 1.570796, 1.682443],accel_mss,speed_ms,0,blend_radius_m)
    |   movel([0.112117, -1.295551, -2.625753, -0.791085, 1.570796, 1.682914],accel_mss,speed_ms,0,blend_radius_m)
    |   movel([0.112419, -1.295641, -2.625700, -0.791048, 1.570796, 1.683215],accel_mss,speed_ms,0,blend_radius_m)
    |   movel([0.111167, -1.297314, -2.624710, -0.790364, 1.570796, 1.681963],accel_mss,speed_ms,0,blend_radius_m)
    |   movel([0.109797, -1.299108, -2.623645, -0.789635, 1.570796, 1.680593],accel_mss,speed_ms,0,blend_radius_m)
    |   movel([0.108182, -1.301220, -2.622386, -0.788783, 1.570796, 1.678978],accel_mss,speed_ms,0,blend_radius_m)
    |   movel([0.106560, -1.303325, -2.621126, -0.787938, 1.570796, 1.677356],accel_mss,speed_ms,0,blend_radius_m)
    |   movel([0.105169, -1.305112, -2.620051, -0.787226, 1.570796, 1.675965],accel_mss,speed_ms,0,blend_radius_m)
    |   movel([0.103939, -1.306679, -2.619105, -0.786605, 1.570796, 1.674736],accel_mss,speed_ms,0,blend_radius_m)
    |   speed_ms = 0.003
    |   movel([0.103813, -1.310267, -2.620648, -0.781474, 1.570796, 1.674610],accel_mss,speed_ms,0,blend_radius_m)
    |   speed_ms = 0.007
    |   movel([0.103818, -1.309935, -2.620849, -0.781604, 1.570796, 1.674615],accel_mss,speed_ms,0,blend_radius_m)
    |   movel([0.104142, -1.309196, -2.621298, -0.781895, 1.570796, 1.674938],accel_mss,speed_ms,0,blend_radius_m)
    |   movel([0.105377, -1.306521, -2.622916, -0.782952, 1.570796, 1.676173],accel_mss,speed_ms,0,blend_radius_m)
    |   movel([0.105952, -1.305264, -2.623673, -0.783452, 1.570796, 1.676748],accel_mss,speed_ms,0,blend_radius_m)
    |   movel([0.106444, -1.304162, -2.624334, -0.783892, 1.570796, 1.677240],accel_mss,speed_ms,0,blend_radius_m)
    |   movel([0.106854, -1.303221, -2.624898, -0.784270, 1.570796, 1.677650],accel_mss,speed_ms,0,blend_radius_m)
    |   movel([0.106834, -1.302859, -2.625115, -0.784415, 1.570796, 1.677630],accel_mss,speed_ms,0,blend_radius_m)
    |   movel([0.106601, -1.302818, -2.625140, -0.784432, 1.570796, 1.677397],accel_mss,speed_ms,0,blend_radius_m)
    |   movel([0.106084, -1.302929, -2.625073, -0.784387, 1.570796, 1.676881],accel_mss,speed_ms,0,blend_radius_m)
    |   movel([0.104894, -1.303295, -2.624854, -0.784240, 1.570796, 1.675691],accel_mss,speed_ms,0,blend_radius_m)
    |   movel([0.104141, -1.303528, -2.624715, -0.784147, 1.570796, 1.674938],accel_mss,speed_ms,0,blend_radius_m)
    |   movel([0.103630, -1.303662, -2.624634, -0.784093, 1.570796, 1.674427],accel_mss,speed_ms,0,blend_radius_m)
    |   movel([0.103281, -1.303731, -2.624593, -0.784065, 1.570796, 1.674077],accel_mss,speed_ms,0,blend_radius_m)
    |   movel([0.103139, -1.303558, -2.624696, -0.784134, 1.570796, 1.673936],accel_mss,speed_ms,0,blend_radius_m)
    |   movel([0.103501, -1.302685, -2.625219, -0.784485, 1.570796, 1.674298],accel_mss,speed_ms,0,blend_radius_m)
    |   movel([0.104030, -1.301482, -2.625938, -0.784970, 1.570796, 1.674826],accel_mss,speed_ms,0,blend_radius_m)
    |   movel([0.104855, -1.299692, -2.627003, -0.785694, 1.570796, 1.675651],accel_mss,speed_ms,0,blend_radius_m)
    |   movel([0.105571, -1.298171, -2.627905, -0.786313, 1.570796, 1.676367],accel_mss,speed_ms,0,blend_radius_m)
    |   movel([0.106206, -1.296848, -2.628687, -0.786854, 1.570796, 1.677002],accel_mss,speed_ms,0,blend_radius_m)
    |   movel([0.106762, -1.295708, -2.629359, -0.787322, 1.570796, 1.677558],accel_mss,speed_ms,0,blend_radius_m)
    |   movel([0.107086, -1.295361, -2.629563, -0.787464, 1.570796, 1.677883],accel_mss,speed_ms,0,blend_radius_m)
    |   movel([0.107542, -1.295166, -2.629678, -0.787545, 1.570796, 1.678339],accel_mss,speed_ms,0,blend_radius_m)
    |   movel([0.108293, -1.294899, -2.629835, -0.787655, 1.570796, 1.679089],accel_mss,speed_ms,0,blend_radius_m)
    |   movel([0.109705, -1.294442, -2.630104, -0.787843, 1.570796, 1.680502],accel_mss,speed_ms,0,blend_radius_m)
    |   movel([0.110994, -1.294039, -2.630340, -0.788010, 1.570796, 1.681790],accel_mss,speed_ms,0,blend_radius_m)
    |   movel([0.111769, -1.293819, -2.630469, -0.788101, 1.570796, 1.682565],accel_mss,speed_ms,0,blend_radius_m)
    |   movel([0.112276, -1.293697, -2.630541, -0.788151, 1.570796, 1.683072],accel_mss,speed_ms,0,blend_radius_m)
    |   movel([0.111888, -1.294693, -2.629956, -0.787740, 1.570796, 1.682685],accel_mss,speed_ms,0,blend_radius_m)
    |   movel([0.111324, -1.295663, -2.629386, -0.787340, 1.570796, 1.682120],accel_mss,speed_ms,0,blend_radius_m)
    |   movel([0.110646, -1.296786, -2.628724, -0.786879, 1.570796, 1.681442],accel_mss,speed_ms,0,blend_radius_m)
    |   movel([0.109696, -1.298348, -2.627800, -0.786241, 1.570796, 1.680492],accel_mss,speed_ms,0,blend_radius_m)
    |   movel([0.109237, -1.299157, -2.627320, -0.785911, 1.570796, 1.680034],accel_mss,speed_ms,0,blend_radius_m)
    |   movel([0.109006, -1.299639, -2.627034, -0.785716, 1.570796, 1.679802],accel_mss,speed_ms,0,blend_radius_m)
    |   movel([0.109167, -1.299855, -2.626906, -0.785628, 1.570796, 1.679964],accel_mss,speed_ms,0,blend_radius_m)
    |   movel([0.109462, -1.299811, -2.626932, -0.785646, 1.570796, 1.680258],accel_mss,speed_ms,0,blend_radius_m)
    |   movel([0.109933, -1.299693, -2.627002, -0.785694, 1.570796, 1.680729],accel_mss,speed_ms,0,blend_radius_m)
    |   movel([0.110719, -1.299452, -2.627145, -0.785791, 1.570796, 1.681516],accel_mss,speed_ms,0,blend_radius_m)
    |   movel([0.111646, -1.299170, -2.627312, -0.785906, 1.570796, 1.682443],accel_mss,speed_ms,0,blend_radius_m)
    |   movel([0.112117, -1.299056, -2.627381, -0.785953, 1.570796, 1.682914],accel_mss,speed_ms,0,blend_radius_m)
    |   movel([0.112419, -1.299145, -2.627327, -0.785916, 1.570796, 1.683215],accel_mss,speed_ms,0,blend_radius_m)
    |   movel([0.111167, -1.300815, -2.626335, -0.785239, 1.570796, 1.681963],accel_mss,speed_ms,0,blend_radius_m)
    |   movel([0.109797, -1.302605, -2.625267, -0.784517, 1.570796, 1.680593],accel_mss,speed_ms,0,blend_radius_m)
    |   movel([0.108182, -1.304712, -2.624004, -0.783673, 1.570796, 1.678978],accel_mss,speed_ms,0,blend_radius_m)
    |   movel([0.106560, -1.306812, -2.622741, -0.782837, 1.570796, 1.677356],accel_mss,speed_ms,0,blend_radius_m)
    |   movel([0.105169, -1.308594, -2.621663, -0.782132, 1.570796, 1.675965],accel_mss,speed_ms,0,blend_radius_m)
    |   movel([0.103939, -1.310158, -2.620714, -0.781517, 1.570796, 1.674736],accel_mss,speed_ms,0,blend_radius_m)
    |   speed_ms = 0.003
    |   movel([0.103813, -1.296516, -2.614163, -0.801711, 1.570796, 1.674610],accel_mss,speed_ms,0,blend_radius_m)
    |   speed_ms = 1.000
    |   movel([0.103813, -1.270306, -2.600804, -0.841279, 1.570796, 1.674610],accel_mss,speed_ms,0,blend_radius_m)
    |   movel([0.097054, -1.268961, -2.601575, -0.841853, 1.570796, 1.667851],accel_mss,speed_ms,0,blend_radius_m)
    |   movel([0.097054, -1.295189, -2.614952, -0.802248, 1.570796, 1.667851],accel_mss,speed_ms,0,blend_radius_m)
    |   speed_ms = 0.003
    |   movel([0.097054, -1.305471, -2.619835, -0.787084, 1.570796, 1.667851],accel_mss,speed_ms,0,blend_radius_m)
    |   speed_ms = 0.007
    |   movel([0.096828, -1.305732, -2.619677, -0.786980, 1.570796, 1.667624],accel_mss,speed_ms,0,blend_radius_m)
    |   movel([0.096502, -1.305914, -2.619567, -0.786908, 1.570796, 1.667298],accel_mss,speed_ms,0,blend_radius_m)
    |   movel([0.095838, -1.306121, -2.619442, -0.786826, 1.570796, 1.666635],accel_mss,speed_ms,0,blend_radius_m)
    |   movel([0.093053, -1.306885, -2.618981, -0.786524, 1.570796, 1.663849],accel_mss,speed_ms,0,blend_radius_m)
    |   movel([0.089387, -1.307997, -2.618307, -0.786085, 1.570796, 1.660183],accel_mss,speed_ms,0,blend_radius_m)
    |   movel([0.085759, -1.309319, -2.617504, -0.785565, 1.570796, 1.656556],accel_mss,speed_ms,0,blend_radius_m)
    |   movel([0.082322, -1.310790, -2.616608, -0.784990, 1.570796, 1.653118],accel_mss,speed_ms,0,blend_radius_m)
    |   movel([0.079223, -1.312346, -2.615658, -0.784385, 1.570796, 1.650019],accel_mss,speed_ms,0,blend_radius_m)
    |   movel([0.076467, -1.313922, -2.614692, -0.783776, 1.570796, 1.647263],accel_mss,speed_ms,0,blend_radius_m)
    |   movel([0.073248, -1.315908, -2.613469, -0.783012, 1.570796, 1.644045],accel_mss,speed_ms,0,blend_radius_m)
    |   movel([0.070195, -1.317895, -2.612241, -0.782253, 1.570796, 1.640991],accel_mss,speed_ms,0,blend_radius_m)
    |   movel([0.068013, -1.319445, -2.611279, -0.781664, 1.570796, 1.638809],accel_mss,speed_ms,0,blend_radius_m)
    |   movel([0.067576, -1.319730, -2.611102, -0.781557, 1.570796, 1.638372],accel_mss,speed_ms,0,blend_radius_m)
    |   movel([0.067261, -1.319825, -2.611043, -0.781521, 1.570796, 1.638057],accel_mss,speed_ms,0,blend_radius_m)
    |   movel([0.066994, -1.319754, -2.611087, -0.781548, 1.570796, 1.637790],accel_mss,speed_ms,0,blend_radius_m)
    |   movel([0.066710, -1.319488, -2.611253, -0.781648, 1.570796, 1.637506],accel_mss,speed_ms,0,blend_radius_m)
    |   movel([0.066534, -1.319145, -2.611466, -0.781778, 1.570796, 1.637330],accel_mss,speed_ms,0,blend_radius_m)
    |   movel([0.066526, -1.318728, -2.611725, -0.781936, 1.570796, 1.637323],accel_mss,speed_ms,0,blend_radius_m)
    |   movel([0.066594, -1.318467, -2.611886, -0.782035, 1.570796, 1.637390],accel_mss,speed_ms,0,blend_radius_m)
    |   movel([0.066867, -1.318064, -2.612136, -0.782189, 1.570796, 1.637663],accel_mss,speed_ms,0,blend_radius_m)
    |   movel([0.067167, -1.317788, -2.612307, -0.782293, 1.570796, 1.637963],accel_mss,speed_ms,0,blend_radius_m)
    |   movel([0.067720, -1.317344, -2.612582, -0.782463, 1.570796, 1.638516],accel_mss,speed_ms,0,blend_radius_m)
    |   movel([0.068900, -1.316468, -2.613124, -0.782797, 1.570796, 1.639696],accel_mss,speed_ms,0,blend_radius_m)
    |   movel([0.070231, -1.315498, -2.613722, -0.783169, 1.570796, 1.641027],accel_mss,speed_ms,0,blend_radius_m)
    |   movel([0.071504, -1.314595, -2.614278, -0.783516, 1.570796, 1.642300],accel_mss,speed_ms,0,blend_radius_m)
    |   movel([0.073287, -1.313443, -2.614985, -0.783960, 1.570796, 1.644084],accel_mss,speed_ms,0,blend_radius_m)
    |   movel([0.076248, -1.311728, -2.616036, -0.784625, 1.570796, 1.647044],accel_mss,speed_ms,0,blend_radius_m)
    |   movel([0.079336, -1.310023, -2.617076, -0.785290, 1.570796, 1.650133],accel_mss,speed_ms,0,blend_radius_m)
    |   movel([0.081717, -1.308817, -2.617810, -0.785763, 1.570796, 1.652514],accel_mss,speed_ms,0,blend_radius_m)
    |   movel([0.083889, -1.307824, -2.618412, -0.786153, 1.570796, 1.654686],accel_mss,speed_ms,0,blend_radius_m)
    |   movel([0.085940, -1.306966, -2.618932, -0.786491, 1.570796, 1.656736],accel_mss,speed_ms,0,blend_radius_m)
    |   movel([0.088113, -1.306152, -2.619424, -0.786813, 1.570796, 1.658909],accel_mss,speed_ms,0,blend_radius_m)
    |   movel([0.090652, -1.305288, -2.619945, -0.787156, 1.570796, 1.661449],accel_mss,speed_ms,0,blend_radius_m)
    |   movel([0.093223, -1.304484, -2.620429, -0.787476, 1.570796, 1.664019],accel_mss,speed_ms,0,blend_radius_m)
    |   movel([0.095145, -1.303969, -2.620739, -0.787681, 1.570796, 1.665941],accel_mss,speed_ms,0,blend_radius_m)
    |   movel([0.096536, -1.303696, -2.620903, -0.787790, 1.570796, 1.667333],accel_mss,speed_ms,0,blend_radius_m)
    |   movel([0.097274, -1.303722, -2.620887, -0.787780, 1.570796, 1.668070],accel_mss,speed_ms,0,blend_radius_m)
    |   movel([0.097500, -1.303897, -2.620782, -0.787710, 1.570796, 1.668297],accel_mss,speed_ms,0,blend_radius_m)
    |   movel([0.097411, -1.304460, -2.620444, -0.787485, 1.570796, 1.668208],accel_mss,speed_ms,0,blend_radius_m)
    |   movel([0.097336, -1.304739, -2.620276, -0.787374, 1.570796, 1.668132],accel_mss,speed_ms,0,blend_radius_m)
    |   movel([0.097240, -1.305028, -2.620101, -0.787259, 1.570796, 1.668037],accel_mss,speed_ms,0,blend_radius_m)
    |   movel([0.097140, -1.305291, -2.619943, -0.787155, 1.570796, 1.667936],accel_mss,speed_ms,0,blend_radius_m)
    |   speed_ms = 0.003
    |   movel([0.097054, -1.308952, -2.621446, -0.781991, 1.570796, 1.667851],accel_mss,speed_ms,0,blend_radius_m)
    |   speed_ms = 0.007
    |   movel([0.096828, -1.309213, -2.621288, -0.781888, 1.570796, 1.667624],accel_mss,speed_ms,0,blend_radius_m)
    |   movel([0.096502, -1.309395, -2.621178, -0.781817, 1.570796, 1.667298],accel_mss,speed_ms,0,blend_radius_m)
    |   movel([0.095838, -1.309601, -2.621052, -0.781735, 1.570796, 1.666635],accel_mss,speed_ms,0,blend_radius_m)
    |   movel([0.093053, -1.310363, -2.620589, -0.781436, 1.570796, 1.663849],accel_mss,speed_ms,0,blend_radius_m)
    |   movel([0.089387, -1.311473, -2.619914, -0.781002, 1.570796, 1.660183],accel_mss,speed_ms,0,blend_radius_m)
    |   movel([0.085759, -1.312792, -2.619109, -0.780488, 1.570796, 1.656556],accel_mss,speed_ms,0,blend_radius_m)
    |   movel([0.082322, -1.314260, -2.618210, -0.779919, 1.570796, 1.653118],accel_mss,speed_ms,0,blend_radius_m)
    |   movel([0.079223, -1.315812, -2.617257, -0.779320, 1.570796, 1.650019],accel_mss,speed_ms,0,blend_radius_m)
    |   movel([0.076467, -1.317384, -2.616288, -0.778717, 1.570796, 1.647263],accel_mss,speed_ms,0,blend_radius_m)
    |   movel([0.073248, -1.319365, -2.615063, -0.777961, 1.570796, 1.644045],accel_mss,speed_ms,0,blend_radius_m)
    |   movel([0.070195, -1.321348, -2.613831, -0.777210, 1.570796, 1.640991],accel_mss,speed_ms,0,blend_radius_m)
    |   movel([0.068013, -1.322894, -2.612867, -0.776628, 1.570796, 1.638809],accel_mss,speed_ms,0,blend_radius_m)
    |   movel([0.067576, -1.323178, -2.612689, -0.776521, 1.570796, 1.638372],accel_mss,speed_ms,0,blend_radius_m)
    |   movel([0.067261, -1.323273, -2.612630, -0.776486, 1.570796, 1.638057],accel_mss,speed_ms,0,blend_radius_m)
    |   movel([0.066994, -1.323202, -2.612674, -0.776512, 1.570796, 1.637790],accel_mss,speed_ms,0,blend_radius_m)
    |   movel([0.066710, -1.322937, -2.612840, -0.776612, 1.570796, 1.637506],accel_mss,speed_ms,0,blend_radius_m)
    |   movel([0.066534, -1.322594, -2.613054, -0.776741, 1.570796, 1.637330],accel_mss,speed_ms,0,blend_radius_m)
    |   movel([0.066526, -1.322178, -2.613314, -0.776897, 1.570796, 1.637323],accel_mss,speed_ms,0,blend_radius_m)
    |   movel([0.066594, -1.321919, -2.613475, -0.776995, 1.570796, 1.637390],accel_mss,speed_ms,0,blend_radius_m)
